# B&R Automation Studio project soft_bellows_plc
Automation Studio 4.9

## Configuration Config1

CPU 4PPC70.0702-20B, AutomationRuntime B4.93, Build 4.1.2, Safety 0.0, Vc V4.72.6

### Task classes (Cpu.sw)
```
Cyclic#1 (cycle 2000 us):
  Server <- Source.UDP.Server.prg
  Client <- Source.UDP.Client.prg
Cyclic#4 (cycle 4000 us, tolerance 80000 us):
  Program1 <- Source.Program.prg
DataObjects: Acp10sys
VcDataObjects: Visu <- Visu.dob
Binaries: FWRules, TCData, udbdef, vccdt, vccbmp, Visu03, vccline, vcfile, arial, vcrt, vccstr, vcbclass, vccbtn, vcmgr, vcgclass, vcdsint, vcptelo, vcchtml, vcpdihd, vcshared, arialbd, vcxml, vccnum, vcpdi855, vccalarm, vccurl, vccslider, vccbar, vcpfppc7, vcctext, Visu01, vcpdsw, vcfntttf, vccovl, vcalarm, Visu02, vcctrend, vcpdi815, vcdsloc, vcchspot, vctcal, vcpk, iomap, arconfig, asfw, ashwac, sysconf, User, Role, ashwd, acp10cfg, Acp10map
Libraries: Acp10man, Acp10par, NcGlobal, Acp10_MC, sys_lib, pomoc_lib, brsystem, runtime, MTLinAlg, AsTCP, AsArLog, traj_lib, regulatory, AsUDP, asstring, standard, astime, fileio, powerlnk, asieccon, vcresman, dataobj
```

### Hardware
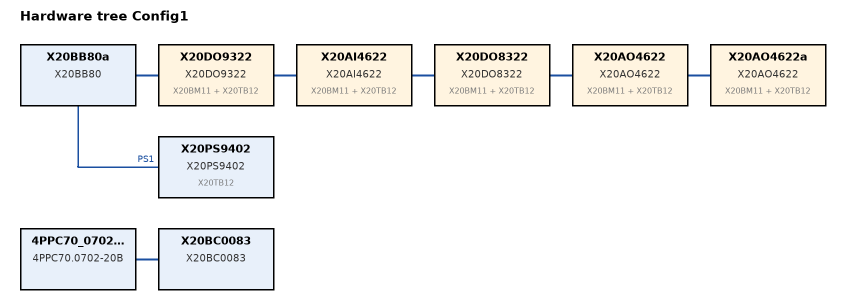
```
4PPC70_0702_20B : 4PPC70.0702-20B v1.5.4.0
  Connector IF2:
    ActivateDevice = 1
    Mode = Manual
    InternetAddress = 192.168.1.100
    SubnetMask = 255.255.255.0
    ActivateSnmp = 2
  ConfigurationID = pneuStand_Config1
  UserPartitionSize = 0
  TimerDeviceType = EPLX2X
  TimerDevice = 4PPC70_0702_20B.IF1
  TaskClassIdleTime = 2000
  Cyclic1Duration = 2000
  Cyclic3Duration = 2000
  Cyclic3Tolerance = 40000
  Cyclic4Duration = 4000
  Cyclic4Tolerance = 80000
  Cyclic5Duration = 20000
  Cyclic5Tolerance = 20000
  Cyclic6Duration = 1000000
  Cyclic6Tolerance = 1000000
  FileDevice1
  FileDeviceName1 = USER
  FileDevicePath1 = USER_PATH
  VcObjectName = Visu
  KeyMatrixPriority = HigherCyclic3
  KeyMappingFile = VC\4PPC70_0702_20B.dis
X20AI4622 : X20AI4622 v1.2.0.0  [SS1 -> X20TB12c.SS; SL -> X20BM11b.SL1]
  Supervision = off
X20AO4622 : X20AO4622 v1.3.0.0  [SS1 -> X20TB12.SS; SL -> X20BM11.SL1]
X20AO4622a : X20AO4622 v1.3.0.0  [SS1 -> X20TB12e.SS; SL -> X20BM11d.SL1]
X20BB80a : X20BB80 v1.1.0.0
X20BC0083 : X20BC0083 v2.14.0.0  [PLK1 -> 4PPC70_0702_20B.IF1 (NodeNumber=1) [Cable Type=PowerlinkCable, Length=10, Version=1.0.0.3]; SL -> X20BB80a.SL1]
  Supervision = off
X20BM11 : X20BM11 v1.1.0.0  [X2X1 -> X20BM11c.X2X2]
X20BM11a : X20BM11 v1.1.0.0  [X2X1 -> X20BB80a.IF1]
X20BM11b : X20BM11 v1.1.0.0  [X2X1 -> X20BM11a.X2X2]
X20BM11c : X20BM11 v1.1.0.0  [X2X1 -> X20BM11b.X2X2]
X20BM11d : X20BM11 v1.1.0.0  [X2X1 -> X20BM11.X2X2]
X20DO8322 : X20DO8322 v1.5.0.0  [SS1 -> X20TB12d.SS; SL -> X20BM11c.SL1]
  Supervision = off
X20DO9322 : X20DO9322 v1.5.0.0  [SS1 -> X20TB12a.SS; SL -> X20BM11a.SL1]
  Supervision = off
X20PS9402 : X20PS9402 v1.2.0.0  [SS1 -> X20TB12b.SS; PS -> X20BB80a.PS1]
  Supervision = off
X20TB12 : X20TB12 v1.0.0.0
X20TB12a : X20TB12 v1.0.0.0
X20TB12b : X20TB12 v1.0.0.0
X20TB12c : X20TB12 v1.0.0.0
X20TB12d : X20TB12 v1.0.0.0
X20TB12e : X20TB12 v1.0.0.0
```

### IoMap.iom - 4PPC70_0702_20B/IoMap.iom
```iecst
VAR_CONFIG
	::tlacidla.ventil[0] AT %QX."X20DO8322".DigitalOutput01;
	::tlacidla.ventil[1] AT %QX."X20DO8322".DigitalOutput02;
	::tlacidla.ventil[2] AT %QX."X20DO8322".DigitalOutput04;
	::tlacidla.ventil[3] AT %QX."X20DO8322".DigitalOutput05;
	::regulatory.reg[1] AT %QW."X20AO4622".AnalogOutput01;
	::regulatory.reg[2] AT %QW."X20AO4622".AnalogOutput02;
	::regulatory.reg[7] AT %QW."X20AO4622".AnalogOutput03;
	::regulatory.reg[6] AT %QW."X20AO4622".AnalogOutput04;
	::regulatory.reg[5] AT %QW."X20AO4622a".AnalogOutput01;
	::regulatory.reg[0] AT %QW."X20AO4622a".AnalogOutput02;
	::regulatory.reg[4] AT %QW."X20AO4622a".AnalogOutput03;
	::regulatory.reg[3] AT %QW."X20AO4622a".AnalogOutput04;
END_VAR
```

## Logical view

Binary libraries used (declarations not repeated): operator, runtime, astime, AsIecCon, Acp10man, Acp10par, NcGlobal, Acp10_MC, sys_lib, brsystem, MTLinAlg 5.12.0, AsArLog, AsTCP, AsUDP, asstring, standard

### Global.typ - Global data types
```iecst
TYPE
	packetUDP : 	STRUCT
		comma : INT; (*Positions of comma in received packet*)
		pStart : INT; (*Start of pressure values*)
		packet_pressure : STRING[80]; (*Full received packet*)
		length : INT; (*Length of full packet*)
		pEnd : INT; (*End of pressure values*)
		pressureString : ARRAY[0..7]OF STRING[8];
		pressureAO : ARRAY[0..7]OF REAL;
	END_STRUCT;
	Analog_input : 	STRUCT
		AI_2 : INT;
		AI_3 : INT;
		AI_4 : INT;
		AI_1 : INT;
	END_STRUCT;
	Digital_output : 	STRUCT
		DO_2 : BOOL;
		DO_3 : BOOL;
		DO_4 : BOOL;
		DO_5 : BOOL;
		DO_6 : BOOL;
		DO_7 : BOOL;
		DO_8 : BOOL;
		DO_9 : BOOL;
		DO_10 : BOOL;
		DO_11 : BOOL;
		DO_12 : BOOL;
		DO_1 : BOOL;
	END_STRUCT;
	regulators : 	STRUCT
		reg_2 : INT;
		reg_3 : INT;
		reg_4 : INT;
		reg_5 : INT;
		reg_6 : INT;
		reg_7 : INT;
		reg_8 : INT;
		reg_1 : INT;
		reg : ARRAY[0..7]OF INT;
	END_STRUCT;
	buttons : 	STRUCT
		zapni : BOOL;
		ventil : ARRAY[0..3]OF BOOL;
	END_STRUCT;
	display_variables : 	STRUCT
		in_reg : ARRAY[0..7]OF INT;
	END_STRUCT;
END_TYPE
```

### Global.var - Global variables
```iecst
VAR
	digital_output : Digital_output;
	tlacidla : buttons;
	regulatory : regulators;
	display : display_variables;
	packet : packetUDP;
	analog_input : Analog_input;
END_VAR
```

### Package Logical/Libraries - Global libraries

### Library Logical/Libraries/traj_lib (ANSIC)

#### traj_lib.typ
```iecst
TYPE
	B_generator_trajektorie_test_T :  STRUCT
		Input1 :  REAL;
		Input2 :  REAL;
		Input3 :  REAL;
		Input4 :  REAL;
		Input :  REAL;
		Gain :  ARRAY[0..299] OF REAL;
		Gain1 :  INT;
	END_STRUCT;

	tag_RTM_generator_trajektorie_T :  STRUCT
		errorStatus :  REFERENCE TO USINT;
		blockIO :  REFERENCE TO B_generator_trajektorie_test_T;
	END_STRUCT;

	RT_MODEL_generator_trajektori_T :tag_RTM_generator_trajektorie_T;	(*  *)

END_TYPE
```

#### generator_trajektorie_test.h
```c
/*
 * generator_trajektorie_test.h
 *
 * Academic License - for use in teaching, academic research, and meeting
 * course requirements at degree granting institutions only.  Not for
 * government, commercial, or other organizational use.
 *
 * Code generation for model "generator_trajektorie_test".
 *
 * Model version              : 1.23
 * Simulink Coder version : 9.6 (R2021b) 14-May-2021
 * C source code generated on : Fri Mar 25 13:28:48 2022
 *
 * Target selection: bur_grt.tlc
 * Note: GRT includes extra infrastructure and instrumentation for prototyping
 * Embedded hardware selection: Intel->x86/Pentium
 * Code generation objectives: Unspecified
 * Validation result: Not run
 */

#ifndef RTW_HEADER_generator_trajektorie_test_h_
#define RTW_HEADER_generator_trajektorie_test_h_
#include <math.h>
#include <stddef.h>
#include <string.h>
#ifndef generator_trajektorie_test_COMMON_INCLUDES_
#define generator_trajektorie_test_COMMON_INCLUDES_
#include <stdlib.h>
#include "rtwtypes.h"
#include "rtw_continuous.h"
#include "rtw_solver.h"
#endif                         /* generator_trajektorie_test_COMMON_INCLUDES_ */

#include "generator_trajektorie_test_types.h"
#include "traj_lib.h"
/* Beginning of Dynamic TypeDefs: */
/* End of Dynamic TypeDefs: */
#ifndef MIN
#define MIN(a,b)	((a) < (b) ? (a) : (b))
#endif

#ifndef MAX
#define MAX(a,b)	((a) > (b) ? (a) : (b))
#endif

#ifndef AST_ROUND
#define AST_ROUND(x) ((x)>=0?(long long)((x)+0.5):(long long)((x)-0.5))
#endif

/* Shared type includes */
#include "multiword_types.h"
#include "rtGetNaN.h"
#include "rt_nonfinite.h"
#include "rtGetInf.h"
#include "rt_defines.h"

/* Macros for accessing real-time model data structure */
#ifndef rtmGetBlockIO
#define rtmGetBlockIO(rtm)             ((rtm)->blockIO)
#endif

#ifndef rtmSetBlockIO
#define rtmSetBlockIO(rtm, val)        ((rtm)->blockIO = (val))
#endif

#ifndef rtmGetErrorStatus
#define rtmGetErrorStatus(rtm)         ((rtm)->errorStatus)
#endif

#ifndef rtmSetErrorStatus
#define rtmSetErrorStatus(rtm, val)    ((rtm)->errorStatus = (val))
#endif

#define generator_trajektorie_test_M_TYPE RT_MODEL_generator_trajektori_T

/* Block signals (default storage) */

/* Real-time Model Data Structure */

/* External data declarations for dependent source files */
extern const char *RT_MEMORY_ALLOCATION_ERROR;

/* Model entry point functions */
extern void generator_trajektorie_test_initializeMemory(RT_MODEL_generator_trajektori_T * const generator_trajektorie_test_M, struct traj* inst);
extern void generator_trajektorie_test_initialize
  (RT_MODEL_generator_trajektori_T *const generator_trajektorie_test_M, struct traj* inst);
extern void generator_trajektorie_test_step(RT_MODEL_generator_trajektori_T *
  const generator_trajektorie_test_M, struct traj* inst);
extern void generator_trajektorie_test_terminate(RT_MODEL_generator_trajektori_T
  * generator_trajektorie_test_M, struct traj* inst);

/*-
 * The generated code includes comments that allow you to trace directly
 * back to the appropriate location in the model.  The basic format
 * is <system>/block_name, where system is the system number (uniquely
 * assigned by Simulink) and block_name is the name of the block.
 *
 * Use the MATLAB hilite_system command to trace the generated code back
 * to the model.  For example,
 *
 * hilite_system('<S3>')    - opens system 3
 * hilite_system('<S3>/Kp') - opens and selects block Kp which resides in S3
 *
 * Here is the system hierarchy for this model
 *
 * '<Root>' : 'generator_trajektorie_test'
 * '<S1>'   : 'generator_trajektorie_test/MATLAB Function'
 */
#endif                            /* RTW_HEADER_generator_trajektorie_test_h_ */
```

#### generator_trajektorie_test_private.h
```c
/*
 * generator_trajektorie_test_private.h
 *
 * Academic License - for use in teaching, academic research, and meeting
 * course requirements at degree granting institutions only.  Not for
 * government, commercial, or other organizational use.
 *
 * Code generation for model "generator_trajektorie_test".
 *
 * Model version              : 1.23
 * Simulink Coder version : 9.6 (R2021b) 14-May-2021
 * C source code generated on : Fri Mar 25 13:28:48 2022
 *
 * Target selection: bur_grt.tlc
 * Note: GRT includes extra infrastructure and instrumentation for prototyping
 * Embedded hardware selection: Intel->x86/Pentium
 * Code generation objectives: Unspecified
 * Validation result: Not run
 */

#ifndef RTW_HEADER_generator_trajektorie_test_private_h_
#define RTW_HEADER_generator_trajektorie_test_private_h_
#include "rtwtypes.h"
#include "multiword_types.h"
#if !defined(rt_VALIDATE_MEMORY)
#define rt_VALIDATE_MEMORY(S, ptr)     if(!(ptr)) {\
 rtmSetErrorStatus(generator_trajektorie_test_M, RT_MEMORY_ALLOCATION_ERROR);\
 }
#endif

#if !defined(rt_FREE)
#if !defined(_WIN32)
#define rt_FREE(ptr)                   if((ptr) != (NULL)) {\
 free((ptr));\
 (ptr) = (NULL);\
 }
#else

/* Visual and other windows compilers declare free without const */
#define rt_FREE(ptr)                   if((ptr) != (NULL)) {\
 free((void *)(ptr));\
 (ptr) = (NULL);\
 }
#endif
#endif
#endif                    /* RTW_HEADER_generator_trajektorie_test_private_h_ */
```

#### generator_trajektorie_test_types.h
```c
/*
 * generator_trajektorie_test_types.h
 *
 * Academic License - for use in teaching, academic research, and meeting
 * course requirements at degree granting institutions only.  Not for
 * government, commercial, or other organizational use.
 *
 * Code generation for model "generator_trajektorie_test".
 *
 * Model version              : 1.23
 * Simulink Coder version : 9.6 (R2021b) 14-May-2021
 * C source code generated on : Fri Mar 25 13:28:48 2022
 *
 * Target selection: bur_grt.tlc
 * Note: GRT includes extra infrastructure and instrumentation for prototyping
 * Embedded hardware selection: Intel->x86/Pentium
 * Code generation objectives: Unspecified
 * Validation result: Not run
 */

#ifndef RTW_HEADER_generator_trajektorie_test_types_h_
#define RTW_HEADER_generator_trajektorie_test_types_h_

/* Model Code Variants */

/* Forward declaration for rtModel */

#endif                      /* RTW_HEADER_generator_trajektorie_test_types_h_ */
```

#### multiword_types.h
```c
/*
 * multiword_types.h
 *
 * Academic License - for use in teaching, academic research, and meeting
 * course requirements at degree granting institutions only.  Not for
 * government, commercial, or other organizational use.
 *
 * Code generation for model "generator_trajektorie_test".
 *
 * Model version              : 1.23
 * Simulink Coder version : 9.6 (R2021b) 14-May-2021
 * C source code generated on : Fri Mar 25 13:28:48 2022
 *
 * Target selection: bur_grt.tlc
 * Note: GRT includes extra infrastructure and instrumentation for prototyping
 * Embedded hardware selection: Intel->x86/Pentium
 * Code generation objectives: Unspecified
 * Validation result: Not run
 */

#ifndef MULTIWORD_TYPES_H
#define MULTIWORD_TYPES_H
#include "rtwtypes.h"

/*
 * MultiWord supporting definitions
 */
typedef long int long_T;

/*
 * MultiWord types
 */
typedef struct {
  uint32_T chunks[2];
} int64m_T;

typedef struct {
  int64m_T re;
  int64m_T im;
} cint64m_T;

typedef struct {
  uint32_T chunks[2];
} uint64m_T;

typedef struct {
  uint64m_T re;
  uint64m_T im;
} cuint64m_T;

typedef struct {
  uint32_T chunks[3];
} int96m_T;

typedef struct {
  int96m_T re;
  int96m_T im;
} cint96m_T;

typedef struct {
  uint32_T chunks[3];
} uint96m_T;

typedef struct {
  uint96m_T re;
  uint96m_T im;
} cuint96m_T;

typedef struct {
  uint32_T chunks[4];
} int128m_T;

typedef struct {
  int128m_T re;
  int128m_T im;
} cint128m_T;

typedef struct {
  uint32_T chunks[4];
} uint128m_T;

typedef struct {
  uint128m_T re;
  uint128m_T im;
} cuint128m_T;

typedef struct {
  uint32_T chunks[5];
} int160m_T;

typedef struct {
  int160m_T re;
  int160m_T im;
} cint160m_T;

typedef struct {
  uint32_T chunks[5];
} uint160m_T;

typedef struct {
  uint160m_T re;
  uint160m_T im;
} cuint160m_T;

typedef struct {
  uint32_T chunks[6];
} int192m_T;

typedef struct {
  int192m_T re;
  int192m_T im;
} cint192m_T;

typedef struct {
  uint32_T chunks[6];
} uint192m_T;

typedef struct {
  uint192m_T re;
  uint192m_T im;
} cuint192m_T;

typedef struct {
  uint32_T chunks[7];
} int224m_T;

typedef struct {
  int224m_T re;
  int224m_T im;
} cint224m_T;

typedef struct {
  uint32_T chunks[7];
} uint224m_T;

typedef struct {
  uint224m_T re;
  uint224m_T im;
} cuint224m_T;

typedef struct {
  uint32_T chunks[8];
} int256m_T;

typedef struct {
  int256m_T re;
  int256m_T im;
} cint256m_T;

typedef struct {
  uint32_T chunks[8];
} uint256m_T;

typedef struct {
  uint256m_T re;
  uint256m_T im;
} cuint256m_T;

typedef struct {
  uint32_T chunks[9];
} int288m_T;

typedef struct {
  int288m_T re;
  int288m_T im;
} cint288m_T;

typedef struct {
  uint32_T chunks[9];
} uint288m_T;

typedef struct {
  uint288m_T re;
  uint288m_T im;
} cuint288m_T;

typedef struct {
  uint32_T chunks[10];
} int320m_T;

typedef struct {
  int320m_T re;
  int320m_T im;
} cint320m_T;

typedef struct {
  uint32_T chunks[10];
} uint320m_T;

typedef struct {
  uint320m_T re;
  uint320m_T im;
} cuint320m_T;

typedef struct {
  uint32_T chunks[11];
} int352m_T;

typedef struct {
  int352m_T re;
  int352m_T im;
} cint352m_T;

typedef struct {
  uint32_T chunks[11];
} uint352m_T;

typedef struct {
  uint352m_T re;
  uint352m_T im;
} cuint352m_T;

typedef struct {
  uint32_T chunks[12];
} int384m_T;

typedef struct {
  int384m_T re;
  int384m_T im;
} cint384m_T;

typedef struct {
  uint32_T chunks[12];
} uint384m_T;

typedef struct {
  uint384m_T re;
  uint384m_T im;
} cuint384m_T;

typedef struct {
  uint32_T chunks[13];
} int416m_T;

typedef struct {
  int416m_T re;
  int416m_T im;
} cint416m_T;

typedef struct {
  uint32_T chunks[13];
} uint416m_T;

typedef struct {
  uint416m_T re;
  uint416m_T im;
} cuint416m_T;

typedef struct {
  uint32_T chunks[14];
} int448m_T;

typedef struct {
  int448m_T re;
  int448m_T im;
} cint448m_T;

typedef struct {
  uint32_T chunks[14];
} uint448m_T;

typedef struct {
  uint448m_T re;
  uint448m_T im;
} cuint448m_T;

typedef struct {
  uint32_T chunks[15];
} int480m_T;

typedef struct {
  int480m_T re;
  int480m_T im;
} cint480m_T;

typedef struct {
  uint32_T chunks[15];
} uint480m_T;

typedef struct {
  uint480m_T re;
  uint480m_T im;
} cuint480m_T;

typedef struct {
  uint32_T chunks[16];
} int512m_T;

typedef struct {
  int512m_T re;
  int512m_T im;
} cint512m_T;

typedef struct {
  uint32_T chunks[16];
} uint512m_T;

typedef struct {
  uint512m_T re;
  uint512m_T im;
} cuint512m_T;

typedef struct {
  uint32_T chunks[17];
} int544m_T;

typedef struct {
  int544m_T re;
  int544m_T im;
} cint544m_T;

typedef struct {
  uint32_T chunks[17];
} uint544m_T;

typedef struct {
  uint544m_T re;
  uint544m_T im;
} cuint544m_T;

typedef struct {
  uint32_T chunks[18];
} int576m_T;

typedef struct {
  int576m_T re;
  int576m_T im;
} cint576m_T;

typedef struct {
  uint32_T chunks[18];
} uint576m_T;

typedef struct {
  uint576m_T re;
  uint576m_T im;
} cuint576m_T;

typedef struct {
  uint32_T chunks[19];
} int608m_T;

typedef struct {
  int608m_T re;
  int608m_T im;
} cint608m_T;

typedef struct {
  uint32_T chunks[19];
} uint608m_T;

typedef struct {
  uint608m_T re;
  uint608m_T im;
} cuint608m_T;

typedef struct {
  uint32_T chunks[20];
} int640m_T;

typedef struct {
  int640m_T re;
  int640m_T im;
} cint640m_T;

typedef struct {
  uint32_T chunks[20];
} uint640m_T;

typedef struct {
  uint640m_T re;
  uint640m_T im;
} cuint640m_T;

typedef struct {
  uint32_T chunks[21];
} int672m_T;

typedef struct {
  int672m_T re;
  int672m_T im;
} cint672m_T;

typedef struct {
  uint32_T chunks[21];
} uint672m_T;

typedef struct {
  uint672m_T re;
  uint672m_T im;
} cuint672m_T;

typedef struct {
  uint32_T chunks[22];
} int704m_T;

typedef struct {
  int704m_T re;
  int704m_T im;
} cint704m_T;

typedef struct {
  uint32_T chunks[22];
} uint704m_T;

typedef struct {
  uint704m_T re;
  uint704m_T im;
} cuint704m_T;

typedef struct {
  uint32_T chunks[23];
} int736m_T;

typedef struct {
  int736m_T re;
  int736m_T im;
} cint736m_T;

typedef struct {
  uint32_T chunks[23];
} uint736m_T;

typedef struct {
  uint736m_T re;
  uint736m_T im;
} cuint736m_T;

typedef struct {
  uint32_T chunks[24];
} int768m_T;

typedef struct {
  int768m_T re;
  int768m_T im;
} cint768m_T;

typedef struct {
  uint32_T chunks[24];
} uint768m_T;

typedef struct {
  uint768m_T re;
  uint768m_T im;
} cuint768m_T;

typedef struct {
  uint32_T chunks[25];
} int800m_T;

typedef struct {
  int800m_T re;
  int800m_T im;
} cint800m_T;

typedef struct {
  uint32_T chunks[25];
} uint800m_T;

typedef struct {
  uint800m_T re;
  uint800m_T im;
} cuint800m_T;

typedef struct {
  uint32_T chunks[26];
} int832m_T;

typedef struct {
  int832m_T re;
  int832m_T im;
} cint832m_T;

typedef struct {
  uint32_T chunks[26];
} uint832m_T;

typedef struct {
  uint832m_T re;
  uint832m_T im;
} cuint832m_T;

typedef struct {
  uint32_T chunks[27];
} int864m_T;

typedef struct {
  int864m_T re;
  int864m_T im;
} cint864m_T;

typedef struct {
  uint32_T chunks[27];
} uint864m_T;

typedef struct {
  uint864m_T re;
  uint864m_T im;
} cuint864m_T;

typedef struct {
  uint32_T chunks[28];
} int896m_T;

typedef struct {
  int896m_T re;
  int896m_T im;
} cint896m_T;

typedef struct {
  uint32_T chunks[28];
} uint896m_T;

typedef struct {
  uint896m_T re;
  uint896m_T im;
} cuint896m_T;

typedef struct {
  uint32_T chunks[29];
} int928m_T;

typedef struct {
  int928m_T re;
  int928m_T im;
} cint928m_T;

typedef struct {
  uint32_T chunks[29];
} uint928m_T;

typedef struct {
  uint928m_T re;
  uint928m_T im;
} cuint928m_T;

typedef struct {
  uint32_T chunks[30];
} int960m_T;

typedef struct {
  int960m_T re;
  int960m_T im;
} cint960m_T;

typedef struct {
  uint32_T chunks[30];
} uint960m_T;

typedef struct {
  uint960m_T re;
  uint960m_T im;
} cuint960m_T;

typedef struct {
  uint32_T chunks[31];
} int992m_T;

typedef struct {
  int992m_T re;
  int992m_T im;
} cint992m_T;

typedef struct {
  uint32_T chunks[31];
} uint992m_T;

typedef struct {
  uint992m_T re;
  uint992m_T im;
} cuint992m_T;

typedef struct {
  uint32_T chunks[32];
} int1024m_T;

typedef struct {
  int1024m_T re;
  int1024m_T im;
} cint1024m_T;

typedef struct {
  uint32_T chunks[32];
} uint1024m_T;

typedef struct {
  uint1024m_T re;
  uint1024m_T im;
} cuint1024m_T;

typedef struct {
  uint32_T chunks[33];
} int1056m_T;

typedef struct {
  int1056m_T re;
  int1056m_T im;
} cint1056m_T;

typedef struct {
  uint32_T chunks[33];
} uint1056m_T;

typedef struct {
  uint1056m_T re;
  uint1056m_T im;
} cuint1056m_T;

typedef struct {
  uint32_T chunks[34];
} int1088m_T;

typedef struct {
  int1088m_T re;
  int1088m_T im;
} cint1088m_T;

typedef struct {
  uint32_T chunks[34];
} uint1088m_T;

typedef struct {
  uint1088m_T re;
  uint1088m_T im;
} cuint1088m_T;

typedef struct {
  uint32_T chunks[35];
} int1120m_T;

typedef struct {
  int1120m_T re;
  int1120m_T im;
} cint1120m_T;

typedef struct {
  uint32_T chunks[35];
} uint1120m_T;

typedef struct {
  uint1120m_T re;
  uint1120m_T im;
} cuint1120m_T;

typedef struct {
  uint32_T chunks[36];
} int1152m_T;

typedef struct {
  int1152m_T re;
  int1152m_T im;
} cint1152m_T;

typedef struct {
  uint32_T chunks[36];
} uint1152m_T;

typedef struct {
  uint1152m_T re;
  uint1152m_T im;
} cuint1152m_T;

typedef struct {
  uint32_T chunks[37];
} int1184m_T;

typedef struct {
  int1184m_T re;
  int1184m_T im;
} cint1184m_T;

typedef struct {
  uint32_T chunks[37];
} uint1184m_T;

typedef struct {
  uint1184m_T re;
  uint1184m_T im;
} cuint1184m_T;

typedef struct {
  uint32_T chunks[38];
} int1216m_T;

typedef struct {
  int1216m_T re;
  int1216m_T im;
} cint1216m_T;

typedef struct {
  uint32_T chunks[38];
} uint1216m_T;

typedef struct {
  uint1216m_T re;
  uint1216m_T im;
} cuint1216m_T;

typedef struct {
  uint32_T chunks[39];
} int1248m_T;

typedef struct {
  int1248m_T re;
  int1248m_T im;
} cint1248m_T;

typedef struct {
  uint32_T chunks[39];
} uint1248m_T;

typedef struct {
  uint1248m_T re;
  uint1248m_T im;
} cuint1248m_T;

typedef struct {
  uint32_T chunks[40];
} int1280m_T;

typedef struct {
  int1280m_T re;
  int1280m_T im;
} cint1280m_T;

typedef struct {
  uint32_T chunks[40];
} uint1280m_T;

typedef struct {
  uint1280m_T re;
  uint1280m_T im;
} cuint1280m_T;

typedef struct {
  uint32_T chunks[41];
} int1312m_T;

typedef struct {
  int1312m_T re;
  int1312m_T im;
} cint1312m_T;

typedef struct {
  uint32_T chunks[41];
} uint1312m_T;

typedef struct {
  uint1312m_T re;
  uint1312m_T im;
} cuint1312m_T;

typedef struct {
  uint32_T chunks[42];
} int1344m_T;

typedef struct {
  int1344m_T re;
  int1344m_T im;
} cint1344m_T;

typedef struct {
  uint32_T chunks[42];
} uint1344m_T;

typedef struct {
  uint1344m_T re;
  uint1344m_T im;
} cuint1344m_T;

typedef struct {
  uint32_T chunks[43];
} int1376m_T;

typedef struct {
  int1376m_T re;
  int1376m_T im;
} cint1376m_T;

typedef struct {
  uint32_T chunks[43];
} uint1376m_T;

typedef struct {
  uint1376m_T re;
  uint1376m_T im;
} cuint1376m_T;

typedef struct {
  uint32_T chunks[44];
} int1408m_T;

typedef struct {
  int1408m_T re;
  int1408m_T im;
} cint1408m_T;

typedef struct {
  uint32_T chunks[44];
} uint1408m_T;

typedef struct {
  uint1408m_T re;
  uint1408m_T im;
} cuint1408m_T;

typedef struct {
  uint32_T chunks[45];
} int1440m_T;

typedef struct {
  int1440m_T re;
  int1440m_T im;
} cint1440m_T;

typedef struct {
  uint32_T chunks[45];
} uint1440m_T;

typedef struct {
  uint1440m_T re;
  uint1440m_T im;
} cuint1440m_T;

typedef struct {
  uint32_T chunks[46];
} int1472m_T;

typedef struct {
  int1472m_T re;
  int1472m_T im;
} cint1472m_T;

typedef struct {
  uint32_T chunks[46];
} uint1472m_T;

typedef struct {
  uint1472m_T re;
  uint1472m_T im;
} cuint1472m_T;

typedef struct {
  uint32_T chunks[47];
} int1504m_T;

typedef struct {
  int1504m_T re;
  int1504m_T im;
} cint1504m_T;

typedef struct {
  uint32_T chunks[47];
} uint1504m_T;

typedef struct {
  uint1504m_T re;
  uint1504m_T im;
} cuint1504m_T;

typedef struct {
  uint32_T chunks[48];
} int1536m_T;

typedef struct {
  int1536m_T re;
  int1536m_T im;
} cint1536m_T;

typedef struct {
  uint32_T chunks[48];
} uint1536m_T;

typedef struct {
  uint1536m_T re;
  uint1536m_T im;
} cuint1536m_T;

typedef struct {
  uint32_T chunks[49];
} int1568m_T;

typedef struct {
  int1568m_T re;
  int1568m_T im;
} cint1568m_T;

typedef struct {
  uint32_T chunks[49];
} uint1568m_T;

typedef struct {
  uint1568m_T re;
  uint1568m_T im;
} cuint1568m_T;

typedef struct {
  uint32_T chunks[50];
} int1600m_T;

typedef struct {
  int1600m_T re;
  int1600m_T im;
} cint1600m_T;

typedef struct {
  uint32_T chunks[50];
} uint1600m_T;

typedef struct {
  uint1600m_T re;
  uint1600m_T im;
} cuint1600m_T;

typedef struct {
  uint32_T chunks[51];
} int1632m_T;

typedef struct {
  int1632m_T re;
  int1632m_T im;
} cint1632m_T;

typedef struct {
  uint32_T chunks[51];
} uint1632m_T;

typedef struct {
  uint1632m_T re;
  uint1632m_T im;
} cuint1632m_T;

typedef struct {
  uint32_T chunks[52];
} int1664m_T;

typedef struct {
  int1664m_T re;
  int1664m_T im;
} cint1664m_T;

typedef struct {
  uint32_T chunks[52];
} uint1664m_T;

typedef struct {
  uint1664m_T re;
  uint1664m_T im;
} cuint1664m_T;

typedef struct {
  uint32_T chunks[53];
} int1696m_T;

typedef struct {
  int1696m_T re;
  int1696m_T im;
} cint1696m_T;

typedef struct {
  uint32_T chunks[53];
} uint1696m_T;

typedef struct {
  uint1696m_T re;
  uint1696m_T im;
} cuint1696m_T;

typedef struct {
  uint32_T chunks[54];
} int1728m_T;

typedef struct {
  int1728m_T re;
  int1728m_T im;
} cint1728m_T;

typedef struct {
  uint32_T chunks[54];
} uint1728m_T;

typedef struct {
  uint1728m_T re;
  uint1728m_T im;
} cuint1728m_T;

typedef struct {
  uint32_T chunks[55];
} int1760m_T;

typedef struct {
  int1760m_T re;
  int1760m_T im;
} cint1760m_T;

typedef struct {
  uint32_T chunks[55];
} uint1760m_T;

typedef struct {
  uint1760m_T re;
  uint1760m_T im;
} cuint1760m_T;

typedef struct {
  uint32_T chunks[56];
} int1792m_T;

typedef struct {
  int1792m_T re;
  int1792m_T im;
} cint1792m_T;

typedef struct {
  uint32_T chunks[56];
} uint1792m_T;

typedef struct {
  uint1792m_T re;
  uint1792m_T im;
} cuint1792m_T;

typedef struct {
  uint32_T chunks[57];
} int1824m_T;

typedef struct {
  int1824m_T re;
  int1824m_T im;
} cint1824m_T;

typedef struct {
  uint32_T chunks[57];
} uint1824m_T;

typedef struct {
  uint1824m_T re;
  uint1824m_T im;
} cuint1824m_T;

typedef struct {
  uint32_T chunks[58];
} int1856m_T;

typedef struct {
  int1856m_T re;
  int1856m_T im;
} cint1856m_T;

typedef struct {
  uint32_T chunks[58];
} uint1856m_T;

typedef struct {
  uint1856m_T re;
  uint1856m_T im;
} cuint1856m_T;

typedef struct {
  uint32_T chunks[59];
} int1888m_T;

typedef struct {
  int1888m_T re;
  int1888m_T im;
} cint1888m_T;

typedef struct {
  uint32_T chunks[59];
} uint1888m_T;

typedef struct {
  uint1888m_T re;
  uint1888m_T im;
} cuint1888m_T;

typedef struct {
  uint32_T chunks[60];
} int1920m_T;

typedef struct {
  int1920m_T re;
  int1920m_T im;
} cint1920m_T;

typedef struct {
  uint32_T chunks[60];
} uint1920m_T;

typedef struct {
  uint1920m_T re;
  uint1920m_T im;
} cuint1920m_T;

typedef struct {
  uint32_T chunks[61];
} int1952m_T;

typedef struct {
  int1952m_T re;
  int1952m_T im;
} cint1952m_T;

typedef struct {
  uint32_T chunks[61];
} uint1952m_T;

typedef struct {
  uint1952m_T re;
  uint1952m_T im;
} cuint1952m_T;

typedef struct {
  uint32_T chunks[62];
} int1984m_T;

typedef struct {
  int1984m_T re;
  int1984m_T im;
} cint1984m_T;

typedef struct {
  uint32_T chunks[62];
} uint1984m_T;

typedef struct {
  uint1984m_T re;
  uint1984m_T im;
} cuint1984m_T;

typedef struct {
  uint32_T chunks[63];
} int2016m_T;

typedef struct {
  int2016m_T re;
  int2016m_T im;
} cint2016m_T;

typedef struct {
  uint32_T chunks[63];
} uint2016m_T;

typedef struct {
  uint2016m_T re;
  uint2016m_T im;
} cuint2016m_T;

typedef struct {
  uint32_T chunks[64];
} int2048m_T;

typedef struct {
  int2048m_T re;
  int2048m_T im;
} cint2048m_T;

typedef struct {
  uint32_T chunks[64];
} uint2048m_T;

typedef struct {
  uint2048m_T re;
  uint2048m_T im;
} cuint2048m_T;

#endif                                 /* MULTIWORD_TYPES_H */
```

#### rt_defines.h
```c
/*
 * rt_defines.h
 *
 * Academic License - for use in teaching, academic research, and meeting
 * course requirements at degree granting institutions only.  Not for
 * government, commercial, or other organizational use.
 *
 * Code generation for model "generator_trajektorie_test".
 *
 * Model version              : 1.23
 * Simulink Coder version : 9.6 (R2021b) 14-May-2021
 * C source code generated on : Fri Mar 25 13:28:48 2022
 *
 * Target selection: bur_grt.tlc
 * Note: GRT includes extra infrastructure and instrumentation for prototyping
 * Embedded hardware selection: Intel->x86/Pentium
 * Code generation objectives: Unspecified
 * Validation result: Not run
 */

#ifndef RTW_HEADER_rt_defines_h_
#define RTW_HEADER_rt_defines_h_

/*===========*
 * Constants *
 *===========*/
#define RT_PI                          3.14159265358979323846
#define RT_PIF                         3.1415927F
#define RT_LN_10                       2.30258509299404568402
#define RT_LN_10F                      2.3025851F
#define RT_LOG10E                      0.43429448190325182765
#define RT_LOG10EF                     0.43429449F
#define RT_E                           2.7182818284590452354
#define RT_EF                          2.7182817F

/*
 * UNUSED_PARAMETER(x)
 *   Used to specify that a function parameter (argument) is required but not
 *   accessed by the function body.
 */
#ifndef UNUSED_PARAMETER
#if defined(__LCC__)
#define UNUSED_PARAMETER(x)                                      /* do nothing */
#else

/*
 * This is the semi-ANSI standard way of indicating that an
 * unused function parameter is required.
 */
#define UNUSED_PARAMETER(x)            (void) (x)
#endif
#endif
#endif                                 /* RTW_HEADER_rt_defines_h_ */
```

#### rtGetInf.h
```c
/*
 * rtGetInf.h
 *
 * Academic License - for use in teaching, academic research, and meeting
 * course requirements at degree granting institutions only.  Not for
 * government, commercial, or other organizational use.
 *
 * Code generation for model "generator_trajektorie_test".
 *
 * Model version              : 1.23
 * Simulink Coder version : 9.6 (R2021b) 14-May-2021
 * C source code generated on : Fri Mar 25 13:28:48 2022
 *
 * Target selection: bur_grt.tlc
 * Note: GRT includes extra infrastructure and instrumentation for prototyping
 * Embedded hardware selection: Intel->x86/Pentium
 * Code generation objectives: Unspecified
 * Validation result: Not run
 */

#ifndef RTW_HEADER_rtGetInf_h_
#define RTW_HEADER_rtGetInf_h_
#include <stddef.h>
#include "rtwtypes.h"
#include "rt_nonfinite.h"

extern real_T rtGetInf(void);
extern real32_T rtGetInfF(void);
extern real_T rtGetMinusInf(void);
extern real32_T rtGetMinusInfF(void);

#endif                                 /* RTW_HEADER_rtGetInf_h_ */
```

#### rtmodel.h
```c
/*
 *  rtmodel.h:
 *
 * Academic License - for use in teaching, academic research, and meeting
 * course requirements at degree granting institutions only.  Not for
 * government, commercial, or other organizational use.
 *
 * Code generation for model "generator_trajektorie_test".
 *
 * Model version              : 1.3
 * Simulink Coder version : 9.6 (R2021b) 14-May-2021
 * C source code generated on : Wed Mar  2 13:13:15 2022
 *
 * Target selection: bur_grt.tlc
 * Note: GRT includes extra infrastructure and instrumentation for prototyping
 * Embedded hardware selection: Intel->x86/Pentium
 * Code generation objectives: Unspecified
 * Validation result: Not run
 */

#ifndef RTW_HEADER_rtmodel_h_
#define RTW_HEADER_rtmodel_h_

/*
 *  Includes the appropriate headers when we are using rtModel
 */
#include "generator_trajektorie_test.h"
#define GRTINTERFACE                   0

/*
 * ROOT_IO_FORMAT: 0 (Individual arguments)
 * ROOT_IO_FORMAT: 1 (Structure reference)
 * ROOT_IO_FORMAT: 2 (Part of model data structure)
 */
#define ROOT_IO_FORMAT                 2

/* Macros generated for backwards compatibility  */
#ifndef rtmGetStopRequested
#define rtmGetStopRequested(rtm)       ((void*) 0)
#endif
#endif                                 /* RTW_HEADER_rtmodel_h_ */
```

#### lib_properties.txt
```
For manual assignment to hardware configuration please
add the following additional include directories:

\Logical\MATLAB_includes\R2021b\

And the following additional build options:

-lm -D RT_MALLOC -D MODEL=generator_trajektorie_test -D NUMST=1 -D NCSTATES=0 -D HAVESTDIO -D RT -D USE_RTMODEL -D CLASSIC_INTERFACE=0 -D ALLOCATIONFCN=1 -D TID01EQ=0 -D MAT_FILE=0 -D ONESTEPFCN=1 -D TERMFCN=1 -D MULTI_INSTANCE_CODE=1 -D INTEGER_CODE=0 -D MT=0
```

#### rtGetNaN.c
```c
/*
 * rtGetNaN.c
 *
 * Academic License - for use in teaching, academic research, and meeting
 * course requirements at degree granting institutions only.  Not for
 * government, commercial, or other organizational use.
 *
 * Code generation for model "generator_trajektorie_test".
 *
 * Model version              : 1.23
 * Simulink Coder version : 9.6 (R2021b) 14-May-2021
 * C source code generated on : Fri Mar 25 13:28:48 2022
 *
 * Target selection: bur_grt.tlc
 * Note: GRT includes extra infrastructure and instrumentation for prototyping
 * Embedded hardware selection: Intel->x86/Pentium
 * Code generation objectives: Unspecified
 * Validation result: Not run
 */

/*
 * Abstract:
 *      Function to initialize non-finite, NaN
 */
#include "rtGetNaN.h"
#define NumBitsPerChar                 8U

/*
 * Initialize rtNaN needed by the generated code.
 * NaN is initialized as non-signaling. Assumes IEEE.
 */
real_T rtGetNaN(void)
{
  size_t bitsPerReal = sizeof(real_T) * (NumBitsPerChar);
  real_T nan = 0.0;
  if (bitsPerReal == 32U) {
    nan = rtGetNaNF();
  } else {
    uint16_T one = 1U;
    enum {
      LittleEndian,
      BigEndian
    } machByteOrder = (*((uint8_T *) &one) == 1U) ? LittleEndian : BigEndian;
    switch (machByteOrder) {
     case LittleEndian:
      {
        union {
          LittleEndianIEEEDouble bitVal;
          real_T fltVal;
        } tmpVal;

        tmpVal.bitVal.words.wordH = 0xFFF80000U;
        tmpVal.bitVal.words.wordL = 0x00000000U;
        nan = tmpVal.fltVal;
        break;
      }

     case BigEndian:
      {
        union {
          BigEndianIEEEDouble bitVal;
          real_T fltVal;
        } tmpVal;

        tmpVal.bitVal.words.wordH = 0x7FFFFFFFU;
        tmpVal.bitVal.words.wordL = 0xFFFFFFFFU;
        nan = tmpVal.fltVal;
        break;
      }
    }
  }

  return nan;
}

/*
 * Initialize rtNaNF needed by the generated code.
 * NaN is initialized as non-signaling. Assumes IEEE.
 */
real32_T rtGetNaNF(void)
{
  IEEESingle nanF = { { 0.0F } };

  uint16_T one = 1U;
  enum {
    LittleEndian,
    BigEndian
  } machByteOrder = (*((uint8_T *) &one) == 1U) ? LittleEndian : BigEndian;
  switch (machByteOrder) {
   case LittleEndian:
    {
      nanF.wordL.wordLuint = 0xFFC00000U;
      break;
    }

   case BigEndian:
    {
      nanF.wordL.wordLuint = 0x7FFFFFFFU;
      break;
    }
  }

  return nanF.wordL.wordLreal;
}
```

### Library Logical/Libraries/pomoc_lib (ANSIC, version 1.00.0)

#### cyklovac_BB_private.h
```c
/*
 * cyklovac_BB_private.h
 *
 * Academic License - for use in teaching, academic research, and meeting
 * course requirements at degree granting institutions only.  Not for
 * government, commercial, or other organizational use.
 *
 * Code generation for model "cyklovac_BB".
 *
 * Model version              : 1.8
 * Simulink Coder version : 9.6 (R2021b) 14-May-2021
 * C source code generated on : Thu Mar 17 07:18:42 2022
 *
 * Target selection: bur_grt.tlc
 * Note: GRT includes extra infrastructure and instrumentation for prototyping
 * Embedded hardware selection: Intel->x86/Pentium
 * Code generation objectives: Unspecified
 * Validation result: Not run
 */

#ifndef RTW_HEADER_cyklovac_BB_private_h_
#define RTW_HEADER_cyklovac_BB_private_h_
#include "rtwtypes.h"
#include "multiword_types.h"
#if !defined(rt_VALIDATE_MEMORY)
#define rt_VALIDATE_MEMORY(S, ptr)     if(!(ptr)) {\
 rtmSetErrorStatus(cyklovac_BB_M, RT_MEMORY_ALLOCATION_ERROR);\
 }
#endif

#if !defined(rt_FREE)
#if !defined(_WIN32)
#define rt_FREE(ptr)                   if((ptr) != (NULL)) {\
 free((ptr));\
 (ptr) = (NULL);\
 }
#else

/* Visual and other windows compilers declare free without const */
#define rt_FREE(ptr)                   if((ptr) != (NULL)) {\
 free((void *)(ptr));\
 (ptr) = (NULL);\
 }
#endif
#endif
#endif                                 /* RTW_HEADER_cyklovac_BB_private_h_ */
```

#### cyklovac_b.c
```c
/********************************************************************
 * COPYRIGHT -- B&R Industrial Automation GmbH
 ********************************************************************
 * Program: pomoc_lib
 * File: pomoc_lib.c
 * Author: MartinV
 * Last modified by: MartinV
 * Created: 17-Mar-2022 07:18:45
 * Last modified: Thu Mar 17 07:18:38 2022
 * Model Version: 1.8
 * Description:
 * modified Comment:
 ********************************************************************
 * Implementation of program pomoc_lib
 ********************************************************************
 * Generated with B&R Automation Studio Target for Simulink V6.5
 * (GRT based)
 ********************************************************************/

#include <bur/plctypes.h>

#include "rtwtypes.h"
#include "rtmodel.h"

#define EXPAND_CONCAT(name1,name2) name1 ## name2
#define CONCAT(name1,name2) EXPAND_CONCAT(name1,name2)
#define RT_MODEL            CONCAT(MODEL,_rtModel)

#ifdef __cplusplus

extern "C" {

#endif

/* Defines */
#define SS_TERMINATE 4
#define SS_OUTPUT 3
#define SS_INITIALIZE 2

#ifdef __cplusplus

}

#endif

#ifdef __cplusplus
    unsigned long bur_heap_size = 6553500;
#endif

void cyklovac_b(struct cyklovac_b* inst)
{
  tag_RTM_cyklovac_BB_T* const cyklovac_BB_M = &(inst)->bur_cyklovac_BB;
	inst->bur_cyklovac_BB.blockIO = &(inst)->bur_B_cyklovac_BB_T;

  switch (inst->ssMethodType)
  {
    case SS_INITIALIZE:

      /* call model initialize functions */
		/*memInit function */
		cyklovac_BB_initializeMemory(cyklovac_BB_M, inst);
		cyklovac_BB_initialize(cyklovac_BB_M, inst);
      break;

    case SS_OUTPUT:
      /* call model step functions */
		cyklovac_BB_step(cyklovac_BB_M, inst);
      break;

    case SS_TERMINATE:
      /* call model terminate function */
		cyklovac_BB_terminate(cyklovac_BB_M, inst);
	  break;
  }
}

/*****************************************************************************
   Function block sample time: 0.008
 *****************************************************************************/

/*****************************************************************************
   B&R Automation Studio Target for Simulink Version: V6.5.1 (03-Dec-2021)
 *****************************************************************************/
```

#### pomoc_lib.typ
```iecst
TYPE
B_cyklovac_BB_T : STRUCT
	Input : REAL;
	Gain : REAL;
	Gain1 : REAL;
	Gain2 : REAL;
END_STRUCT;
ConstP_cyklovac_BB_T : STRUCT
	Constant_Value : ARRAY[0..2351] OF LREAL;
END_STRUCT;
tag_RTM_cyklovac_BB_T : STRUCT
	errorStatus : REFERENCE TO USINT;
	blockIO : REFERENCE TO B_cyklovac_BB_T;
END_STRUCT;
RT_MODEL_cyklovac_BB_T : tag_RTM_cyklovac_BB_T;

END_TYPE
TYPE
END_TYPE
```

#### rt_defines.h
```c
/*
 * rt_defines.h
 *
 * Academic License - for use in teaching, academic research, and meeting
 * course requirements at degree granting institutions only.  Not for
 * government, commercial, or other organizational use.
 *
 * Code generation for model "cyklovac_BB".
 *
 * Model version              : 1.8
 * Simulink Coder version : 9.6 (R2021b) 14-May-2021
 * C source code generated on : Thu Mar 17 07:18:42 2022
 *
 * Target selection: bur_grt.tlc
 * Note: GRT includes extra infrastructure and instrumentation for prototyping
 * Embedded hardware selection: Intel->x86/Pentium
 * Code generation objectives: Unspecified
 * Validation result: Not run
 */

#ifndef RTW_HEADER_rt_defines_h_
#define RTW_HEADER_rt_defines_h_

/*===========*
 * Constants *
 *===========*/
#define RT_PI                          3.14159265358979323846
#define RT_PIF                         3.1415927F
#define RT_LN_10                       2.30258509299404568402
#define RT_LN_10F                      2.3025851F
#define RT_LOG10E                      0.43429448190325182765
#define RT_LOG10EF                     0.43429449F
#define RT_E                           2.7182818284590452354
#define RT_EF                          2.7182817F

/*
 * UNUSED_PARAMETER(x)
 *   Used to specify that a function parameter (argument) is required but not
 *   accessed by the function body.
 */
#ifndef UNUSED_PARAMETER
#if defined(__LCC__)
#define UNUSED_PARAMETER(x)                                      /* do nothing */
#else

/*
 * This is the semi-ANSI standard way of indicating that an
 * unused function parameter is required.
 */
#define UNUSED_PARAMETER(x)            (void) (x)
#endif
#endif
#endif                                 /* RTW_HEADER_rt_defines_h_ */
```

#### rtmodel.h
```c
/*
 *  rtmodel.h:
 *
 * Academic License - for use in teaching, academic research, and meeting
 * course requirements at degree granting institutions only.  Not for
 * government, commercial, or other organizational use.
 *
 * Code generation for model "cyklovac_BB".
 *
 * Model version              : 1.8
 * Simulink Coder version : 9.6 (R2021b) 14-May-2021
 * C source code generated on : Thu Mar 17 07:18:42 2022
 *
 * Target selection: bur_grt.tlc
 * Note: GRT includes extra infrastructure and instrumentation for prototyping
 * Embedded hardware selection: Intel->x86/Pentium
 * Code generation objectives: Unspecified
 * Validation result: Not run
 */

#ifndef RTW_HEADER_rtmodel_h_
#define RTW_HEADER_rtmodel_h_

/*
 *  Includes the appropriate headers when we are using rtModel
 */
#include "cyklovac_BB.h"
#define GRTINTERFACE                   0

/*
 * ROOT_IO_FORMAT: 0 (Individual arguments)
 * ROOT_IO_FORMAT: 1 (Structure reference)
 * ROOT_IO_FORMAT: 2 (Part of model data structure)
 */
#define ROOT_IO_FORMAT                 2

/* Macros generated for backwards compatibility  */
#ifndef rtmGetStopRequested
#define rtmGetStopRequested(rtm)       ((void*) 0)
#endif
#endif                                 /* RTW_HEADER_rtmodel_h_ */
```

#### rtwtypes.h
```c
/*
 * rtwtypes.h
 *
 * Academic License - for use in teaching, academic research, and meeting
 * course requirements at degree granting institutions only.  Not for
 * government, commercial, or other organizational use.
 *
 * Code generation for model "cyklovac_BB".
 *
 * Model version              : 1.8
 * Simulink Coder version : 9.6 (R2021b) 14-May-2021
 * C source code generated on : Thu Mar 17 07:18:42 2022
 *
 * Target selection: bur_grt.tlc
 * Note: GRT includes extra infrastructure and instrumentation for prototyping
 * Embedded hardware selection: Intel->x86/Pentium
 * Code generation objectives: Unspecified
 * Validation result: Not run
 */

#ifndef RTWTYPES_H
#define RTWTYPES_H
#include "tmwtypes.h"
#ifndef POINTER_T
#define POINTER_T

typedef void * pointer_T;

#endif

/* Logical type definitions */
#if (!defined(__cplusplus))
#ifndef false
#define false                          (0U)
#endif

#ifndef true
#define true                           (1U)
#endif
#endif
#endif                                 /* RTWTYPES_H */
```

### Library Logical/Libraries/regulatory (ANSIC, version 1.00.0)

#### reg_FF_PI_pl_regr_stiff.h
```c
/*
 * reg_FF_PI_pl_regr_stiff.h
 *
 * Academic License - for use in teaching, academic research, and meeting
 * course requirements at degree granting institutions only.  Not for
 * government, commercial, or other organizational use.
 *
 * Code generation for model "reg_FF_PI_pl_regr_stiff".
 *
 * Model version              : 1.135
 * Simulink Coder version : 9.6 (R2021b) 14-May-2021
 * C source code generated on : Tue Sep 27 10:51:43 2022
 *
 * Target selection: bur_grt.tlc
 * Note: GRT includes extra infrastructure and instrumentation for prototyping
 * Embedded hardware selection: Intel->x86/Pentium
 * Code generation objectives: Unspecified
 * Validation result: Not run
 */

#ifndef RTW_HEADER_reg_FF_PI_pl_regr_stiff_h_
#define RTW_HEADER_reg_FF_PI_pl_regr_stiff_h_
#include <math.h>
#include <stddef.h>
#include <string.h>
#ifndef reg_FF_PI_pl_regr_stiff_COMMON_INCLUDES_
#define reg_FF_PI_pl_regr_stiff_COMMON_INCLUDES_
#include <stdlib.h>
#include "rtwtypes.h"
#include "rtw_continuous.h"
#include "rtw_solver.h"
#endif                            /* reg_FF_PI_pl_regr_stiff_COMMON_INCLUDES_ */

#include "reg_FF_PI_pl_regr_stiff_types.h"
#include "regulatory.h"
/* Beginning of Dynamic TypeDefs: */
/* End of Dynamic TypeDefs: */
#ifndef MIN
#define MIN(a,b)	((a) < (b) ? (a) : (b))
#endif

#ifndef MAX
#define MAX(a,b)	((a) > (b) ? (a) : (b))
#endif

#ifndef AST_ROUND
#define AST_ROUND(x) ((x)>=0?(long long)((x)+0.5):(long long)((x)-0.5))
#endif

/* Shared type includes */
#include "multiword_types.h"

/* Macros for accessing real-time model data structure */
#ifndef rtmGetBlockIO
#define rtmGetBlockIO(rtm)             ((rtm)->blockIO)
#endif

#ifndef rtmSetBlockIO
#define rtmSetBlockIO(rtm, val)        ((rtm)->blockIO = (val))
#endif

#ifndef rtmGetRootDWork
#define rtmGetRootDWork(rtm)           ((rtm)->dwork)
#endif

#ifndef rtmSetRootDWork
#define rtmSetRootDWork(rtm, val)      ((rtm)->dwork = (val))
#endif

#ifndef rtmGetErrorStatus
#define rtmGetErrorStatus(rtm)         ((rtm)->errorStatus)
#endif

#ifndef rtmSetErrorStatus
#define rtmSetErrorStatus(rtm, val)    ((rtm)->errorStatus = (val))
#endif

#define reg_FF_PI_pl_regr_stiff_M_TYPE RT_MODEL_reg_FF_PI_pl_regr_st_T

/* Block signals (default storage) */

/* Block states (default storage) for system '<Root>' */

/* Constant parameters (default storage) */

/* Real-time Model Data Structure */

/* External data declarations for dependent source files */
extern const char *RT_MEMORY_ALLOCATION_ERROR;

/* Constant parameters (default storage) */
extern const ConstP_reg_FF_PI_pl_regr_stif_T reg_FF_PI_pl_regr_stiff_ConstP;

/* Model entry point functions */
extern void reg_FF_PI_pl_regr_stiff_initializeMemory(RT_MODEL_reg_FF_PI_pl_regr_st_T * const reg_FF_PI_pl_regr_stiff_M, struct FF_PID_r_t* inst);
extern void reg_FF_PI_pl_regr_stiff_initialize(RT_MODEL_reg_FF_PI_pl_regr_st_T *
  const reg_FF_PI_pl_regr_stiff_M, struct FF_PID_r_t* inst);
extern void reg_FF_PI_pl_regr_stiff_step(RT_MODEL_reg_FF_PI_pl_regr_st_T *const
  reg_FF_PI_pl_regr_stiff_M, struct FF_PID_r_t* inst);
extern void reg_FF_PI_pl_regr_stiff_terminate(RT_MODEL_reg_FF_PI_pl_regr_st_T
  * reg_FF_PI_pl_regr_stiff_M, struct FF_PID_r_t* inst);

/*-
 * The generated code includes comments that allow you to trace directly
 * back to the appropriate location in the model.  The basic format
 * is <system>/block_name, where system is the system number (uniquely
 * assigned by Simulink) and block_name is the name of the block.
 *
 * Use the MATLAB hilite_system command to trace the generated code back
 * to the model.  For example,
 *
 * hilite_system('<S3>')    - opens system 3
 * hilite_system('<S3>/Kp') - opens and selects block Kp which resides in S3
 *
 * Here is the system hierarchy for this model
 *
 * '<Root>' : 'reg_FF_PI_pl_regr_stiff'
 * '<S1>'   : 'reg_FF_PI_pl_regr_stiff/FF_zlozka'
 * '<S2>'   : 'reg_FF_PI_pl_regr_stiff/Subsystem'
 * '<S3>'   : 'reg_FF_PI_pl_regr_stiff/FF_zlozka/MATLAB Function'
 * '<S4>'   : 'reg_FF_PI_pl_regr_stiff/Subsystem/AlfaX_baseY2deltaz2'
 * '<S5>'   : 'reg_FF_PI_pl_regr_stiff/Subsystem/V_PID_Yellow'
 * '<S6>'   : 'reg_FF_PI_pl_regr_stiff/Subsystem/V_PID_Yellow1'
 * '<S7>'   : 'reg_FF_PI_pl_regr_stiff/Subsystem/V_PID_blue'
 * '<S8>'   : 'reg_FF_PI_pl_regr_stiff/Subsystem/abs2relat1'
 * '<S9>'   : 'reg_FF_PI_pl_regr_stiff/Subsystem/abs2relat2'
 * '<S10>'  : 'reg_FF_PI_pl_regr_stiff/Subsystem/abs2relat3'
 * '<S11>'  : 'reg_FF_PI_pl_regr_stiff/Subsystem/abs2relat4'
 * '<S12>'  : 'reg_FF_PI_pl_regr_stiff/Subsystem/abs2relat7'
 * '<S13>'  : 'reg_FF_PI_pl_regr_stiff/Subsystem/abs2relat8'
 * '<S14>'  : 'reg_FF_PI_pl_regr_stiff/Subsystem/AlfaX_baseY2deltaz2/requested alfa 2 deltaz1'
 * '<S15>'  : 'reg_FF_PI_pl_regr_stiff/Subsystem/V_PID_Yellow/Anti-windup'
 * '<S16>'  : 'reg_FF_PI_pl_regr_stiff/Subsystem/V_PID_Yellow/D Gain'
 * '<S17>'  : 'reg_FF_PI_pl_regr_stiff/Subsystem/V_PID_Yellow/Filter'
 * '<S18>'  : 'reg_FF_PI_pl_regr_stiff/Subsystem/V_PID_Yellow/Filter ICs'
 * '<S19>'  : 'reg_FF_PI_pl_regr_stiff/Subsystem/V_PID_Yellow/I Gain'
 * '<S20>'  : 'reg_FF_PI_pl_regr_stiff/Subsystem/V_PID_Yellow/Ideal P Gain'
 * '<S21>'  : 'reg_FF_PI_pl_regr_stiff/Subsystem/V_PID_Yellow/Ideal P Gain Fdbk'
 * '<S22>'  : 'reg_FF_PI_pl_regr_stiff/Subsystem/V_PID_Yellow/Integrator'
 * '<S23>'  : 'reg_FF_PI_pl_regr_stiff/Subsystem/V_PID_Yellow/Integrator ICs'
 * '<S24>'  : 'reg_FF_PI_pl_regr_stiff/Subsystem/V_PID_Yellow/N Copy'
 * '<S25>'  : 'reg_FF_PI_pl_regr_stiff/Subsystem/V_PID_Yellow/N Gain'
 * '<S26>'  : 'reg_FF_PI_pl_regr_stiff/Subsystem/V_PID_Yellow/P Copy'
 * '<S27>'  : 'reg_FF_PI_pl_regr_stiff/Subsystem/V_PID_Yellow/Parallel P Gain'
 * '<S28>'  : 'reg_FF_PI_pl_regr_stiff/Subsystem/V_PID_Yellow/Reset Signal'
 * '<S29>'  : 'reg_FF_PI_pl_regr_stiff/Subsystem/V_PID_Yellow/Saturation'
 * '<S30>'  : 'reg_FF_PI_pl_regr_stiff/Subsystem/V_PID_Yellow/Saturation Fdbk'
 * '<S31>'  : 'reg_FF_PI_pl_regr_stiff/Subsystem/V_PID_Yellow/Sum'
 * '<S32>'  : 'reg_FF_PI_pl_regr_stiff/Subsystem/V_PID_Yellow/Sum Fdbk'
 * '<S33>'  : 'reg_FF_PI_pl_regr_stiff/Subsystem/V_PID_Yellow/Tracking Mode'
 * '<S34>'  : 'reg_FF_PI_pl_regr_stiff/Subsystem/V_PID_Yellow/Tracking Mode Sum'
 * '<S35>'  : 'reg_FF_PI_pl_regr_stiff/Subsystem/V_PID_Yellow/Tsamp - Integral'
 * '<S36>'  : 'reg_FF_PI_pl_regr_stiff/Subsystem/V_PID_Yellow/Tsamp - Ngain'
 * '<S37>'  : 'reg_FF_PI_pl_regr_stiff/Subsystem/V_PID_Yellow/postSat Signal'
 * '<S38>'  : 'reg_FF_PI_pl_regr_stiff/Subsystem/V_PID_Yellow/preSat Signal'
 * '<S39>'  : 'reg_FF_PI_pl_regr_stiff/Subsystem/V_PID_Yellow/Anti-windup/Passthrough'
 * '<S40>'  : 'reg_FF_PI_pl_regr_stiff/Subsystem/V_PID_Yellow/D Gain/External Parameters'
 * '<S41>'  : 'reg_FF_PI_pl_regr_stiff/Subsystem/V_PID_Yellow/Filter/Disc. Forward Euler Filter'
 * '<S42>'  : 'reg_FF_PI_pl_regr_stiff/Subsystem/V_PID_Yellow/Filter ICs/Internal IC - Filter'
 * '<S43>'  : 'reg_FF_PI_pl_regr_stiff/Subsystem/V_PID_Yellow/I Gain/External Parameters'
 * '<S44>'  : 'reg_FF_PI_pl_regr_stiff/Subsystem/V_PID_Yellow/Ideal P Gain/Passthrough'
 * '<S45>'  : 'reg_FF_PI_pl_regr_stiff/Subsystem/V_PID_Yellow/Ideal P Gain Fdbk/Disabled'
 * '<S46>'  : 'reg_FF_PI_pl_regr_stiff/Subsystem/V_PID_Yellow/Integrator/Discrete'
 * '<S47>'  : 'reg_FF_PI_pl_regr_stiff/Subsystem/V_PID_Yellow/Integrator ICs/Internal IC'
 * '<S48>'  : 'reg_FF_PI_pl_regr_stiff/Subsystem/V_PID_Yellow/N Copy/Disabled'
 * '<S49>'  : 'reg_FF_PI_pl_regr_stiff/Subsystem/V_PID_Yellow/N Gain/External Parameters'
 * '<S50>'  : 'reg_FF_PI_pl_regr_stiff/Subsystem/V_PID_Yellow/P Copy/Disabled'
 * '<S51>'  : 'reg_FF_PI_pl_regr_stiff/Subsystem/V_PID_Yellow/Parallel P Gain/External Parameters'
 * '<S52>'  : 'reg_FF_PI_pl_regr_stiff/Subsystem/V_PID_Yellow/Reset Signal/External Reset'
 * '<S53>'  : 'reg_FF_PI_pl_regr_stiff/Subsystem/V_PID_Yellow/Saturation/External'
 * '<S54>'  : 'reg_FF_PI_pl_regr_stiff/Subsystem/V_PID_Yellow/Saturation/External/Saturation Dynamic'
 * '<S55>'  : 'reg_FF_PI_pl_regr_stiff/Subsystem/V_PID_Yellow/Saturation Fdbk/Disabled'
 * '<S56>'  : 'reg_FF_PI_pl_regr_stiff/Subsystem/V_PID_Yellow/Sum/Sum_PID'
 * '<S57>'  : 'reg_FF_PI_pl_regr_stiff/Subsystem/V_PID_Yellow/Sum Fdbk/Disabled'
 * '<S58>'  : 'reg_FF_PI_pl_regr_stiff/Subsystem/V_PID_Yellow/Tracking Mode/Disabled'
 * '<S59>'  : 'reg_FF_PI_pl_regr_stiff/Subsystem/V_PID_Yellow/Tracking Mode Sum/Passthrough'
 * '<S60>'  : 'reg_FF_PI_pl_regr_stiff/Subsystem/V_PID_Yellow/Tsamp - Integral/Passthrough'
 * '<S61>'  : 'reg_FF_PI_pl_regr_stiff/Subsystem/V_PID_Yellow/Tsamp - Ngain/Passthrough'
 * '<S62>'  : 'reg_FF_PI_pl_regr_stiff/Subsystem/V_PID_Yellow/postSat Signal/Forward_Path'
 * '<S63>'  : 'reg_FF_PI_pl_regr_stiff/Subsystem/V_PID_Yellow/preSat Signal/Forward_Path'
 * '<S64>'  : 'reg_FF_PI_pl_regr_stiff/Subsystem/V_PID_Yellow1/Anti-windup'
 * '<S65>'  : 'reg_FF_PI_pl_regr_stiff/Subsystem/V_PID_Yellow1/D Gain'
 * '<S66>'  : 'reg_FF_PI_pl_regr_stiff/Subsystem/V_PID_Yellow1/Filter'
 * '<S67>'  : 'reg_FF_PI_pl_regr_stiff/Subsystem/V_PID_Yellow1/Filter ICs'
 * '<S68>'  : 'reg_FF_PI_pl_regr_stiff/Subsystem/V_PID_Yellow1/I Gain'
 * '<S69>'  : 'reg_FF_PI_pl_regr_stiff/Subsystem/V_PID_Yellow1/Ideal P Gain'
 * '<S70>'  : 'reg_FF_PI_pl_regr_stiff/Subsystem/V_PID_Yellow1/Ideal P Gain Fdbk'
 * '<S71>'  : 'reg_FF_PI_pl_regr_stiff/Subsystem/V_PID_Yellow1/Integrator'
 * '<S72>'  : 'reg_FF_PI_pl_regr_stiff/Subsystem/V_PID_Yellow1/Integrator ICs'
 * '<S73>'  : 'reg_FF_PI_pl_regr_stiff/Subsystem/V_PID_Yellow1/N Copy'
 * '<S74>'  : 'reg_FF_PI_pl_regr_stiff/Subsystem/V_PID_Yellow1/N Gain'
 * '<S75>'  : 'reg_FF_PI_pl_regr_stiff/Subsystem/V_PID_Yellow1/P Copy'
 * '<S76>'  : 'reg_FF_PI_pl_regr_stiff/Subsystem/V_PID_Yellow1/Parallel P Gain'
 * '<S77>'  : 'reg_FF_PI_pl_regr_stiff/Subsystem/V_PID_Yellow1/Reset Signal'
 * '<S78>'  : 'reg_FF_PI_pl_regr_stiff/Subsystem/V_PID_Yellow1/Saturation'
 * '<S79>'  : 'reg_FF_PI_pl_regr_stiff/Subsystem/V_PID_Yellow1/Saturation Fdbk'
 * '<S80>'  : 'reg_FF_PI_pl_regr_stiff/Subsystem/V_PID_Yellow1/Sum'
 * '<S81>'  : 'reg_FF_PI_pl_regr_stiff/Subsystem/V_PID_Yellow1/Sum Fdbk'
 * '<S82>'  : 'reg_FF_PI_pl_regr_stiff/Subsystem/V_PID_Yellow1/Tracking Mode'
 * '<S83>'  : 'reg_FF_PI_pl_regr_stiff/Subsystem/V_PID_Yellow1/Tracking Mode Sum'
 * '<S84>'  : 'reg_FF_PI_pl_regr_stiff/Subsystem/V_PID_Yellow1/Tsamp - Integral'
 * '<S85>'  : 'reg_FF_PI_pl_regr_stiff/Subsystem/V_PID_Yellow1/Tsamp - Ngain'
 * '<S86>'  : 'reg_FF_PI_pl_regr_stiff/Subsystem/V_PID_Yellow1/postSat Signal'
 * '<S87>'  : 'reg_FF_PI_pl_regr_stiff/Subsystem/V_PID_Yellow1/preSat Signal'
 * '<S88>'  : 'reg_FF_PI_pl_regr_stiff/Subsystem/V_PID_Yellow1/Anti-windup/Passthrough'
 * '<S89>'  : 'reg_FF_PI_pl_regr_stiff/Subsystem/V_PID_Yellow1/D Gain/External Parameters'
 * '<S90>'  : 'reg_FF_PI_pl_regr_stiff/Subsystem/V_PID_Yellow1/Filter/Disc. Forward Euler Filter'
 * '<S91>'  : 'reg_FF_PI_pl_regr_stiff/Subsystem/V_PID_Yellow1/Filter ICs/Internal IC - Filter'
 * '<S92>'  : 'reg_FF_PI_pl_regr_stiff/Subsystem/V_PID_Yellow1/I Gain/External Parameters'
 * '<S93>'  : 'reg_FF_PI_pl_regr_stiff/Subsystem/V_PID_Yellow1/Ideal P Gain/Passthrough'
 * '<S94>'  : 'reg_FF_PI_pl_regr_stiff/Subsystem/V_PID_Yellow1/Ideal P Gain Fdbk/Disabled'
 * '<S95>'  : 'reg_FF_PI_pl_regr_stiff/Subsystem/V_PID_Yellow1/Integrator/Discrete'
 * '<S96>'  : 'reg_FF_PI_pl_regr_stiff/Subsystem/V_PID_Yellow1/Integrator ICs/Internal IC'
 * '<S97>'  : 'reg_FF_PI_pl_regr_stiff/Subsystem/V_PID_Yellow1/N Copy/Disabled'
 * '<S98>'  : 'reg_FF_PI_pl_regr_stiff/Subsystem/V_PID_Yellow1/N Gain/External Parameters'
 * '<S99>'  : 'reg_FF_PI_pl_regr_stiff/Subsystem/V_PID_Yellow1/P Copy/Disabled'
 * '<S100>' : 'reg_FF_PI_pl_regr_stiff/Subsystem/V_PID_Yellow1/Parallel P Gain/External Parameters'
 * '<S101>' : 'reg_FF_PI_pl_regr_stiff/Subsystem/V_PID_Yellow1/Reset Signal/External Reset'
 * '<S102>' : 'reg_FF_PI_pl_regr_stiff/Subsystem/V_PID_Yellow1/Saturation/External'
 * '<S103>' : 'reg_FF_PI_pl_regr_stiff/Subsystem/V_PID_Yellow1/Saturation/External/Saturation Dynamic'
 * '<S104>' : 'reg_FF_PI_pl_regr_stiff/Subsystem/V_PID_Yellow1/Saturation Fdbk/Disabled'
 * '<S105>' : 'reg_FF_PI_pl_regr_stiff/Subsystem/V_PID_Yellow1/Sum/Sum_PID'
 * '<S106>' : 'reg_FF_PI_pl_regr_stiff/Subsystem/V_PID_Yellow1/Sum Fdbk/Disabled'
 * '<S107>' : 'reg_FF_PI_pl_regr_stiff/Subsystem/V_PID_Yellow1/Tracking Mode/Disabled'
 * '<S108>' : 'reg_FF_PI_pl_regr_stiff/Subsystem/V_PID_Yellow1/Tracking Mode Sum/Passthrough'
 * '<S109>' : 'reg_FF_PI_pl_regr_stiff/Subsystem/V_PID_Yellow1/Tsamp - Integral/Passthrough'
 * '<S110>' : 'reg_FF_PI_pl_regr_stiff/Subsystem/V_PID_Yellow1/Tsamp - Ngain/Passthrough'
 * '<S111>' : 'reg_FF_PI_pl_regr_stiff/Subsystem/V_PID_Yellow1/postSat Signal/Forward_Path'
 * '<S112>' : 'reg_FF_PI_pl_regr_stiff/Subsystem/V_PID_Yellow1/preSat Signal/Forward_Path'
 * '<S113>' : 'reg_FF_PI_pl_regr_stiff/Subsystem/V_PID_blue/Anti-windup'
 * '<S114>' : 'reg_FF_PI_pl_regr_stiff/Subsystem/V_PID_blue/D Gain'
 * '<S115>' : 'reg_FF_PI_pl_regr_stiff/Subsystem/V_PID_blue/Filter'
 * '<S116>' : 'reg_FF_PI_pl_regr_stiff/Subsystem/V_PID_blue/Filter ICs'
 * '<S117>' : 'reg_FF_PI_pl_regr_stiff/Subsystem/V_PID_blue/I Gain'
 * '<S118>' : 'reg_FF_PI_pl_regr_stiff/Subsystem/V_PID_blue/Ideal P Gain'
 * '<S119>' : 'reg_FF_PI_pl_regr_stiff/Subsystem/V_PID_blue/Ideal P Gain Fdbk'
 * '<S120>' : 'reg_FF_PI_pl_regr_stiff/Subsystem/V_PID_blue/Integrator'
 * '<S121>' : 'reg_FF_PI_pl_regr_stiff/Subsystem/V_PID_blue/Integrator ICs'
 * '<S122>' : 'reg_FF_PI_pl_regr_stiff/Subsystem/V_PID_blue/N Copy'
 * '<S123>' : 'reg_FF_PI_pl_regr_stiff/Subsystem/V_PID_blue/N Gain'
 * '<S124>' : 'reg_FF_PI_pl_regr_stiff/Subsystem/V_PID_blue/P Copy'
 * '<S125>' : 'reg_FF_PI_pl_regr_stiff/Subsystem/V_PID_blue/Parallel P Gain'
 * '<S126>' : 'reg_FF_PI_pl_regr_stiff/Subsystem/V_PID_blue/Reset Signal'
 * '<S127>' : 'reg_FF_PI_pl_regr_stiff/Subsystem/V_PID_blue/Saturation'
 * '<S128>' : 'reg_FF_PI_pl_regr_stiff/Subsystem/V_PID_blue/Saturation Fdbk'
 * '<S129>' : 'reg_FF_PI_pl_regr_stiff/Subsystem/V_PID_blue/Sum'
 * '<S130>' : 'reg_FF_PI_pl_regr_stiff/Subsystem/V_PID_blue/Sum Fdbk'
 * '<S131>' : 'reg_FF_PI_pl_regr_stiff/Subsystem/V_PID_blue/Tracking Mode'
 * '<S132>' : 'reg_FF_PI_pl_regr_stiff/Subsystem/V_PID_blue/Tracking Mode Sum'
 * '<S133>' : 'reg_FF_PI_pl_regr_stiff/Subsystem/V_PID_blue/Tsamp - Integral'
 * '<S134>' : 'reg_FF_PI_pl_regr_stiff/Subsystem/V_PID_blue/Tsamp - Ngain'
 * '<S135>' : 'reg_FF_PI_pl_regr_stiff/Subsystem/V_PID_blue/postSat Signal'
 * '<S136>' : 'reg_FF_PI_pl_regr_stiff/Subsystem/V_PID_blue/preSat Signal'
 * '<S137>' : 'reg_FF_PI_pl_regr_stiff/Subsystem/V_PID_blue/Anti-windup/Passthrough'
 * '<S138>' : 'reg_FF_PI_pl_regr_stiff/Subsystem/V_PID_blue/D Gain/External Parameters'
 * '<S139>' : 'reg_FF_PI_pl_regr_stiff/Subsystem/V_PID_blue/Filter/Disc. Forward Euler Filter'
 * '<S140>' : 'reg_FF_PI_pl_regr_stiff/Subsystem/V_PID_blue/Filter ICs/Internal IC - Filter'
 * '<S141>' : 'reg_FF_PI_pl_regr_stiff/Subsystem/V_PID_blue/I Gain/External Parameters'
 * '<S142>' : 'reg_FF_PI_pl_regr_stiff/Subsystem/V_PID_blue/Ideal P Gain/Passthrough'
 * '<S143>' : 'reg_FF_PI_pl_regr_stiff/Subsystem/V_PID_blue/Ideal P Gain Fdbk/Disabled'
 * '<S144>' : 'reg_FF_PI_pl_regr_stiff/Subsystem/V_PID_blue/Integrator/Discrete'
 * '<S145>' : 'reg_FF_PI_pl_regr_stiff/Subsystem/V_PID_blue/Integrator ICs/Internal IC'
 * '<S146>' : 'reg_FF_PI_pl_regr_stiff/Subsystem/V_PID_blue/N Copy/Disabled'
 * '<S147>' : 'reg_FF_PI_pl_regr_stiff/Subsystem/V_PID_blue/N Gain/External Parameters'
 * '<S148>' : 'reg_FF_PI_pl_regr_stiff/Subsystem/V_PID_blue/P Copy/Disabled'
 * '<S149>' : 'reg_FF_PI_pl_regr_stiff/Subsystem/V_PID_blue/Parallel P Gain/External Parameters'
 * '<S150>' : 'reg_FF_PI_pl_regr_stiff/Subsystem/V_PID_blue/Reset Signal/External Reset'
 * '<S151>' : 'reg_FF_PI_pl_regr_stiff/Subsystem/V_PID_blue/Saturation/External'
 * '<S152>' : 'reg_FF_PI_pl_regr_stiff/Subsystem/V_PID_blue/Saturation/External/Saturation Dynamic'
 * '<S153>' : 'reg_FF_PI_pl_regr_stiff/Subsystem/V_PID_blue/Saturation Fdbk/Disabled'
 * '<S154>' : 'reg_FF_PI_pl_regr_stiff/Subsystem/V_PID_blue/Sum/Sum_PID'
 * '<S155>' : 'reg_FF_PI_pl_regr_stiff/Subsystem/V_PID_blue/Sum Fdbk/Disabled'
 * '<S156>' : 'reg_FF_PI_pl_regr_stiff/Subsystem/V_PID_blue/Tracking Mode/Disabled'
 * '<S157>' : 'reg_FF_PI_pl_regr_stiff/Subsystem/V_PID_blue/Tracking Mode Sum/Passthrough'
 * '<S158>' : 'reg_FF_PI_pl_regr_stiff/Subsystem/V_PID_blue/Tsamp - Integral/Passthrough'
 * '<S159>' : 'reg_FF_PI_pl_regr_stiff/Subsystem/V_PID_blue/Tsamp - Ngain/Passthrough'
 * '<S160>' : 'reg_FF_PI_pl_regr_stiff/Subsystem/V_PID_blue/postSat Signal/Forward_Path'
 * '<S161>' : 'reg_FF_PI_pl_regr_stiff/Subsystem/V_PID_blue/preSat Signal/Forward_Path'
 */
#endif                               /* RTW_HEADER_reg_FF_PI_pl_regr_stiff_h_ */
```

#### reg_FF_PI_pl_regr_stiff_data.c
```c
/*
 * reg_FF_PI_pl_regr_stiff_data.c
 *
 * Academic License - for use in teaching, academic research, and meeting
 * course requirements at degree granting institutions only.  Not for
 * government, commercial, or other organizational use.
 *
 * Code generation for model "reg_FF_PI_pl_regr_stiff".
 *
 * Model version              : 1.135
 * Simulink Coder version : 9.6 (R2021b) 14-May-2021
 * C source code generated on : Tue Sep 27 10:51:43 2022
 *
 * Target selection: bur_grt.tlc
 * Note: GRT includes extra infrastructure and instrumentation for prototyping
 * Embedded hardware selection: Intel->x86/Pentium
 * Code generation objectives: Unspecified
 * Validation result: Not run
 */

#include "reg_FF_PI_pl_regr_stiff.h"
#include "reg_FF_PI_pl_regr_stiff_private.h"

/* Constant parameters (default storage) */
const ConstP_reg_FF_PI_pl_regr_stif_T reg_FF_PI_pl_regr_stiff_ConstP = {
  /* Expression: coef_1blue
   * Referenced by: '<S1>/Constant'
   */
  { 0.0017105750782315647, -0.00031894042792665118, 0.00035451787790138196,
    -0.00019972200976834959, -4.3892191255761959E-6, -0.00027272249934474538,
    -0.0090478565722579233, 0.0054482716433918608, -0.0072683292922697922,
    0.00413929721958372, 0.00011303098682474825, 0.005591677047672953,
    -0.16681175073563032, -0.036143207245384182, 0.061165365811016628,
    -0.035360608238866748, -0.0011446751359908019, -0.047290107610719861,
    1.9314414355397496, 0.11599151682470536, -0.27274287157744381,
    0.16106157257347073, 0.0059214601396658942, 0.21348955813855988,
    -8.214194337602315, -0.17468404062406745, 0.6935075165131781,
    -0.42202772508074771, -0.016877335878941583, -0.55515365502246838,
    17.123747629688115, 0.0669008896991383, -1.0026784691064161,
    0.63585828567519109, 0.026421042370275552, 0.831151470907112,
    -16.462934654986736, 0.079274206258717048, 0.76227189768315973,
    -0.50974126037567646, -0.020778480585300123, -0.66377130446245836,
    6.95932519589881, -0.12150704958189475, -0.2350544296785472,
    0.16808162279516273, 0.0063626246901319922, 0.21805719235011847 },

  /* Expression: coef_2green
   * Referenced by: '<S1>/Constant1'
   */
  { -0.00038837768098208894, -0.00065117847140775634, 0.00020964331658933648,
    -0.00018966178503272696, 3.6107136311502476E-5, -0.00024567775366209614,
    0.040858546502079623, 0.013145297264238857, -0.0038628601851493733,
    0.00381104087840559, -0.00078121720792697876, 0.00494457781501693,
    -0.65271977929603131, -0.10904154399504047, 0.029139742826547764,
    -0.031407923824548177, 0.007065116461826647, -0.040866436032779611,
    4.4274857655001005, 0.48099251537940674, -0.11739905582318358,
    0.13731679994241536, -0.034458101183743185, 0.17944913231215021,
    -15.481147119163195, -1.2192478431872231, 0.27498378684430841,
    -0.3438802890129693, 0.0971390050296614, -0.45202364142946455,
    29.093533123706937, 1.7796492959360444, -0.37826210079672062,
    0.49388247912156341, -0.15713393344808899, 0.65356045383838535,
    -26.820653555856456, -1.3767944130597296, 0.30889409220045694,
    -0.37750822598435141, 0.13499544127719082, -0.50254981985427571,
    10.589080614584185, 0.46805035762142011, -0.055008004115544067,
    0.11889561406308008, -0.048021210874138291, 0.15896689069549794 },

  /* Expression: coef_3yellow
   * Referenced by: '<S1>/Constant3'
   */
  { 0.0040655521860770679, -0.00045625459374585214, 0.00039587384671225151,
    -0.00028172651766770795, -6.7214130921795348E-5, -0.00028248251395603281,
    -0.052274548967079511, 0.0084304027358908049, -0.0084374664797956141,
    0.0058331765704457876, 0.0015123649012436069, 0.0056840040026990453,
    0.15271371298337824, -0.062075974257985153, 0.073622574381782768,
    -0.049821467704821772, -0.014136189017056839, -0.0469477448909448,
    0.70330100029796949, 0.2325052510651455, -0.33964790581471743,
    0.22704315289173943, 0.070767737933930264, 0.20592112565908618,
    -5.5665529664061006, -0.46853556022720089, 0.89425321396155255,
    -0.59536150815747069, -0.20361499567782843, -0.51788809106330591,
    13.92427212519536, 0.487773373707155, -1.3442475203161097,
    0.89740396531665878, 0.33491638476311841, 0.7474525928110074,
    -14.331234712148808, -0.20455292310497739, 1.0456791951890665,
    -0.71989856223038, -0.29138519106015026, -0.57384727370638533,
    6.25235418888368, 0.032212696269155724, -0.38388460202577607,
    0.23671769120847469, 0.10374886423005664, 0.18103901615539519 }
};
```

#### reg_FF_PI_pl_regr_stiff_private.h
```c
/*
 * reg_FF_PI_pl_regr_stiff_private.h
 *
 * Academic License - for use in teaching, academic research, and meeting
 * course requirements at degree granting institutions only.  Not for
 * government, commercial, or other organizational use.
 *
 * Code generation for model "reg_FF_PI_pl_regr_stiff".
 *
 * Model version              : 1.135
 * Simulink Coder version : 9.6 (R2021b) 14-May-2021
 * C source code generated on : Tue Sep 27 10:51:43 2022
 *
 * Target selection: bur_grt.tlc
 * Note: GRT includes extra infrastructure and instrumentation for prototyping
 * Embedded hardware selection: Intel->x86/Pentium
 * Code generation objectives: Unspecified
 * Validation result: Not run
 */

#ifndef RTW_HEADER_reg_FF_PI_pl_regr_stiff_private_h_
#define RTW_HEADER_reg_FF_PI_pl_regr_stiff_private_h_
#include "rtwtypes.h"
#include "multiword_types.h"
#if !defined(rt_VALIDATE_MEMORY)
#define rt_VALIDATE_MEMORY(S, ptr)     if(!(ptr)) {\
 rtmSetErrorStatus(reg_FF_PI_pl_regr_stiff_M, RT_MEMORY_ALLOCATION_ERROR);\
 }
#endif

#if !defined(rt_FREE)
#if !defined(_WIN32)
#define rt_FREE(ptr)                   if((ptr) != (NULL)) {\
 free((ptr));\
 (ptr) = (NULL);\
 }
#else

/* Visual and other windows compilers declare free without const */
#define rt_FREE(ptr)                   if((ptr) != (NULL)) {\
 free((void *)(ptr));\
 (ptr) = (NULL);\
 }
#endif
#endif
#endif                       /* RTW_HEADER_reg_FF_PI_pl_regr_stiff_private_h_ */
```

#### reg_FF_PI_pl_regr_stiff_types.h
```c
/*
 * reg_FF_PI_pl_regr_stiff_types.h
 *
 * Academic License - for use in teaching, academic research, and meeting
 * course requirements at degree granting institutions only.  Not for
 * government, commercial, or other organizational use.
 *
 * Code generation for model "reg_FF_PI_pl_regr_stiff".
 *
 * Model version              : 1.135
 * Simulink Coder version : 9.6 (R2021b) 14-May-2021
 * C source code generated on : Tue Sep 27 10:51:43 2022
 *
 * Target selection: bur_grt.tlc
 * Note: GRT includes extra infrastructure and instrumentation for prototyping
 * Embedded hardware selection: Intel->x86/Pentium
 * Code generation objectives: Unspecified
 * Validation result: Not run
 */

#ifndef RTW_HEADER_reg_FF_PI_pl_regr_stiff_types_h_
#define RTW_HEADER_reg_FF_PI_pl_regr_stiff_types_h_

/* Model Code Variants */

/* Forward declaration for rtModel */

#endif                         /* RTW_HEADER_reg_FF_PI_pl_regr_stiff_types_h_ */
```

#### regulatory.typ
```iecst
TYPE
	emxArray_real_T :  STRUCT
		data :  REFERENCE TO LREAL;
		size :  REFERENCE TO DINT;
		allocatedSize :  DINT;
		numDimensions :  DINT;
		canFreeData :  BOOL;
	END_STRUCT;

	B_regulator_FF_PI_T :  STRUCT
		Input1 :  REAL;
		Input2 :  REAL;
		Input3 :  REAL;
		Input4 :  REAL;
		Input11 :  REAL;
		Input5 :  REAL;
		Input13 :  REAL;
		Input14 :  REAL;
		Input8 :  REAL;
		Input9 :  REAL;
		Input10 :  REAL;
		Sum :  REAL;
		Input7 :  REAL;
		Sum2 :  REAL;
		Input6 :  REAL;
		Sum1 :  REAL;
		Input12 :  REAL;
	END_STRUCT;

	DW_regulator_FF_PI_T :  STRUCT
		Integrator_DSTATE :  LREAL;
		Filter_DSTATE :  LREAL;
		Integrator_DSTATE_o :  LREAL;
		Filter_DSTATE_f :  LREAL;
		Integrator_DSTATE_i :  LREAL;
		Filter_DSTATE_a :  LREAL;
		Integrator_PrevResetState :  SINT;
		Filter_PrevResetState :  SINT;
		Integrator_PrevResetState_l :  SINT;
		Filter_PrevResetState_e :  SINT;
		Integrator_PrevResetState_e :  SINT;
		Filter_PrevResetState_h :  SINT;
	END_STRUCT;

	ConstP_regulator_FF_PI_T :  STRUCT
		Constant_Value_m :  ARRAY[0..113] OF REAL;
		Constant1_Value_b :  ARRAY[0..113] OF REAL;
		Constant2_Value :  ARRAY[0..113] OF REAL;
		Constant3_Value :  ARRAY[0..113] OF REAL;
	END_STRUCT;

	tag_RTM_regulator_FF_PI_T :  STRUCT
		errorStatus :  REFERENCE TO USINT;
		blockIO :  REFERENCE TO B_regulator_FF_PI_T;
		dwork :  REFERENCE TO DW_regulator_FF_PI_T;
	END_STRUCT;

	B_regulator_FF_PI_plane_regre_T :  STRUCT
		Input1 :  REAL;
		Input2 :  REAL;
		Input3 :  REAL;
		Input4 :  REAL;
		Input11 :  REAL;
		Input5 :  REAL;
		Input13 :  REAL;
		Input14 :  REAL;
		Sum :  REAL;
		Input7 :  REAL;
		Sum2 :  REAL;
		Input6 :  REAL;
		Sum1 :  REAL;
		Input10 :  REAL;
		Input12 :  REAL;
		Input8 :  REAL;
		Input9 :  REAL;
	END_STRUCT;

	DW_regulator_FF_PI_plane_regr_T :  STRUCT
		Integrator_DSTATE :  LREAL;
		Filter_DSTATE :  LREAL;
		Integrator_DSTATE_o :  LREAL;
		Filter_DSTATE_f :  LREAL;
		Integrator_DSTATE_i :  LREAL;
		Filter_DSTATE_a :  LREAL;
		Integrator_PrevResetState :  SINT;
		Filter_PrevResetState :  SINT;
		Integrator_PrevResetState_l :  SINT;
		Filter_PrevResetState_e :  SINT;
		Integrator_PrevResetState_e :  SINT;
		Filter_PrevResetState_h :  SINT;
	END_STRUCT;

	tag_RTM_regulator_FF_PI_plane_T :  STRUCT
		errorStatus :  REFERENCE TO USINT;
		blockIO :  REFERENCE TO B_regulator_FF_PI_plane_regre_T;
		dwork :  REFERENCE TO DW_regulator_FF_PI_plane_regr_T;
	END_STRUCT;

	B_PID_constant_T :  STRUCT
		Input1 :  REAL;
		Input2 :  REAL;
		Input3 :  REAL;
		Input4 :  REAL;
		Input11 :  REAL;
		Input5 :  REAL;
		Input13 :  REAL;
		Input14 :  REAL;
		Switch2 :  REAL;
		Input6 :  REAL;
		Switch1 :  REAL;
		Input7 :  REAL;
		Switch :  REAL;
		Input12 :  REAL;
	END_STRUCT;

	DW_PID_constant_T :  STRUCT
		Integrator_DSTATE :  LREAL;
		Filter_DSTATE :  LREAL;
		Integrator_DSTATE_f :  LREAL;
		Filter_DSTATE_j :  LREAL;
		Integrator_DSTATE_h :  LREAL;
		Filter_DSTATE_m :  LREAL;
		Integrator_PrevResetState :  SINT;
		Filter_PrevResetState :  SINT;
		Integrator_PrevResetState_m :  SINT;
		Filter_PrevResetState_e :  SINT;
		Integrator_PrevResetState_l :  SINT;
		Filter_PrevResetState_k :  SINT;
	END_STRUCT;

	tag_RTM_PID_constant_T :  STRUCT
		errorStatus :  REFERENCE TO USINT;
		blockIO :  REFERENCE TO B_PID_constant_T;
		dwork :  REFERENCE TO DW_PID_constant_T;
	END_STRUCT;

	B_requestedalfa2deltaz1_reg_F_T :  STRUCT
		Blue_real :  REAL;
		Green_real :  REAL;
		Yellow_real :  REAL;
		Blue_ref :  REAL;
		Green_ref :  REAL;
		Yellow_ref :  REAL;
	END_STRUCT;

	B_regulator_nelin_P_T :  STRUCT
		Input1 :  REAL;
		Input2 :  REAL;
		Input3 :  REAL;
		Input4 :  REAL;
		Gain7 :  REAL;
		Gain9 :  REAL;
		Gain8 :  REAL;
	END_STRUCT;

	tag_RTM_regulator_nelin_P_T :  STRUCT
		errorStatus :  REFERENCE TO USINT;
		blockIO :  REFERENCE TO B_regulator_nelin_P_T;
	END_STRUCT;

	B_PID_co_T :  STRUCT
		Input1 :  REAL;
		Input2 :  REAL;
		Input3 :  REAL;
		Input4 :  REAL;
		Input11 :  REAL;
		Input5 :  REAL;
		Input13 :  REAL;
		Input14 :  REAL;
		Switch2 :  REAL;
		Input6 :  REAL;
		Switch1 :  REAL;
		Input7 :  REAL;
		Switch :  REAL;
		Input12 :  REAL;
	END_STRUCT;

	DW_PID_co_T :  STRUCT
		Integrator_DSTATE :  LREAL;
		Filter_DSTATE :  LREAL;
		Integrator_DSTATE_f :  LREAL;
		Filter_DSTATE_j :  LREAL;
		Integrator_DSTATE_h :  LREAL;
		Filter_DSTATE_m :  LREAL;
		Integrator_PrevResetState :  SINT;
		Filter_PrevResetState :  SINT;
		Integrator_PrevResetState_m :  SINT;
		Filter_PrevResetState_e :  SINT;
		Integrator_PrevResetState_l :  SINT;
		Filter_PrevResetState_k :  SINT;
	END_STRUCT;

	tag_RTM_PID_co_T :  STRUCT
		errorStatus :  REFERENCE TO USINT;
		blockIO :  REFERENCE TO B_PID_co_T;
		dwork :  REFERENCE TO DW_PID_co_T;
	END_STRUCT;

	B_reg_FF_PI_pl_regr_stiff_T :  STRUCT
		Input15 :  REAL;
		Input1 :  REAL;
		Input2 :  REAL;
		Input3 :  REAL;
		Input4 :  REAL;
		Input11 :  REAL;
		Input5 :  REAL;
		Input13 :  REAL;
		Input14 :  REAL;
		Sum :  REAL;
		Input7 :  REAL;
		Sum2 :  REAL;
		Input6 :  REAL;
		Sum1 :  REAL;
		Input10 :  REAL;
		Input12 :  REAL;
		Input8 :  REAL;
		Input9 :  REAL;
	END_STRUCT;

	DW_reg_FF_PI_pl_regr_stiff_T :  STRUCT
		Integrator_DSTATE :  LREAL;
		Filter_DSTATE :  LREAL;
		Integrator_DSTATE_o :  LREAL;
		Filter_DSTATE_f :  LREAL;
		Integrator_DSTATE_i :  LREAL;
		Filter_DSTATE_a :  LREAL;
		Integrator_PrevResetState :  SINT;
		Filter_PrevResetState :  SINT;
		Integrator_PrevResetState_l :  SINT;
		Filter_PrevResetState_e :  SINT;
		Integrator_PrevResetState_e :  SINT;
		Filter_PrevResetState_h :  SINT;
	END_STRUCT;

	ConstP_reg_FF_PI_pl_regr_stif_T :  STRUCT
		Constant_Value :  ARRAY[0..47] OF LREAL;
		Constant1_Value :  ARRAY[0..47] OF LREAL;
		Constant3_Value :  ARRAY[0..47] OF LREAL;
	END_STRUCT;

	tag_RTM_reg_FF_PI_pl_regr_sti_T :  STRUCT
		errorStatus :  REFERENCE TO USINT;
		blockIO :  REFERENCE TO B_reg_FF_PI_pl_regr_stiff_T;
		dwork :  REFERENCE TO DW_reg_FF_PI_pl_regr_stiff_T;
	END_STRUCT;

	emxArray_real_T_regulator_FF_T2 :emxArray_real_T;	(*  *)

	RT_MODEL_regulator_FF_PI_T :tag_RTM_regulator_FF_PI_T;	(*  *)

	RT_MODEL_regulator_FF_PI_plan_T :tag_RTM_regulator_FF_PI_plane_T;	(*  *)

	RT_MODEL_PID_constant_T :tag_RTM_PID_constant_T;	(*  *)

	RT_MODEL_regulator_nelin_P_T :tag_RTM_regulator_nelin_P_T;	(*  *)

	RT_MODEL_PID_co_T :tag_RTM_PID_co_T;	(*  *)

	RT_MODEL_reg_FF_PI_pl_regr_st_T :tag_RTM_reg_FF_PI_pl_regr_sti_T;	(*  *)

END_TYPE
```

### Program Logical/Source/Program (IEC)

#### Cyclic.st
```iecst
PROGRAM _CYCLIC

	IF tlacidla.zapni=TRUE THEN

		FOR i:=0 TO 7 BY 1 DO
			regulatory.reg[i] := REAL_TO_INT(display.in_reg[i]/100*32765/9);
		END_FOR

	ELSE

		FOR i:=0 TO 3 BY 1 DO
			tlacidla.ventil[i] := FALSE;
		END_FOR

		FOR i:=0 TO 7 BY 1 DO
			regulatory.reg[i] := 0;
		END_FOR

	END_IF

END_PROGRAM
```

#### Init.st
```iecst
PROGRAM _INIT
	(* Insert code here *)

END_PROGRAM
```

### LibAsUDP1_ST.typ
```iecst
(********************************************************************
 * COPYRIGHT -- Bernecker + Rainer
 ********************************************************************
 * File: Global.typ
 * Author: Bernecker + Rainer
 * Created: June 02, 2008
 ********************************************************************
 * Global data types of project LibAsUDP
 ********************************************************************)

TYPE
	LibAsUDP1_ST_typ : 	STRUCT  (*Datatyp for global Variables*)
		receive_data : ARRAY[0..100] OF UDINT; (*Data which has been received*)
		send_data : ARRAY[0..100] OF UDINT; (*Data which should be sent*)
	END_STRUCT;
END_TYPE
```

### Program Logical/Source/UDP/Client

#### Client.st
```iecst
(********************************************************************
 * COPYRIGHT -- Bernecker + Rainer
 ********************************************************************
 * Program: Client
 * File: Client.st
 * Author: Bernecker + Rainer
 * Created: June 02, 2008
 ********************************************************************
 * Implementation of program Client
 ********************************************************************)

PROGRAM _CYCLIC

	LibAsUDP1_ST.send_data[0] := LibAsUDP1_ST.send_data[0] + 1;  (* Generate a "running" variable for Data transfer *)

	CASE Client.sStep OF

		0:	(* Open UDP Port *)
			Client.UdpOpen_0.enable := 1;
			Client.UdpOpen_0.pIfAddr := 0;	(* Listen on all TCP/IP Interfaces*)
			Client.UdpOpen_0.port := 12051;	(* Port to listen*)
			Client.UdpOpen_0.options := 0;
			Client.UdpOpen_0;	(* Call the Function*)

			IF Client.UdpOpen_0.status = 0 THEN  (* UdpOpen successful*)
				Client.sStep := 1;
			ELSIF Client.UdpOpen_0.status = ERR_FUB_BUSY THEN  (* UdpOpen not finished -> redo *)
			  (* Busy *)
			ELSE  (* Goto Error Step *)
				Client.sStep := 10;
			END_IF

		1:	(* Send Data to the Server *)
			Client.server_address := '192.168.1.506';	(* IP Address of the Server *)
			Client.server_portnumber := 12050;	(* Port number of the Server *)

			Client.UdpSend_0.enable := 1;
			Client.UdpSend_0.ident := Client.UdpOpen_0.ident;	(* Connection Ident from AsUDP.UDP_Open *)
			Client.UdpSend_0.pHost := ADR(Client.server_address);
			Client.UdpSend_0.port := Client.server_portnumber;
			Client.UdpSend_0.pData := ADR(LibAsUDP1_ST.send_data);	(* Which data to send *)
			Client.UdpSend_0.datalen := SIZEOF(LibAsUDP1_ST.send_data);	(* Lenght of data to send *)
			Client.UdpSend_0.flags := 0;
			Client.UdpSend_0;	(* Call the Function*)

			IF Client.UdpSend_0.status = 0 THEN  (* Data sent *)
				Client.sStep := 2;
			ELSIF Client.UdpSend_0.status = ERR_FUB_BUSY THEN  (* UdpSend not finished -> redo *)
			  (* Busy *)
			ELSE  (* Goto Error Step *)
				Client.sStep := 10;
			END_IF

		2:	(* Receive Data from the Server *)
			Client.UdpRecv_0.enable := 1;
			Client.UdpRecv_0.ident := Client.UdpOpen_0.ident;  (* Connection Ident from AsUDP.UDP_Open *)
			Client.UdpRecv_0.pData	:= ADR(LibAsUDP1_ST.receive_data);  (* Where to store the incoming data *)
			Client.UdpRecv_0.datamax := SIZEOF(LibAsUDP1_ST.receive_data);  (* Lenght of data buffer *)
			Client.UdpRecv_0.flags := 0;
			Client.UdpRecv_0;  (* Call the Function*)

			IF Client.UdpRecv_0.status = 0 THEN  (* Data was received successfully -> Send next packet *)
				Client.sStep := 3;
				Client.no_data_received_count := 0;
			ELSIF Client.UdpRecv_0.status = udpERR_NO_DATA THEN  (* No data received - wait *)
			  (* No Data received *)
			  	Client.no_data_received_count := Client.no_data_received_count + 1;	(* Increase if no data are received *)

				IF Client.no_data_received_count > 200 THEN		(* No data timeout for TC1 [10ms] *)
					Client.no_data_received_count := 0;
					Client.sStep := 1;	(* Send again *)
				END_IF
			ELSIF Client.UdpRecv_0.status = ERR_FUB_BUSY THEN  (* UdpRecv not finished -> redo *)
			  (* Busy *)
			ELSE  (* Goto Error Step *)
				Client.sStep := 10;
			END_IF

		3: (* Close connection *)
			Client.UdpClose_0.enable := 1;
			Client.UdpClose_0.ident := Client.UdpOpen_0.ident;  (* Connection Ident from AsUDP.UDP_Open *)
			Client.UdpClose_0;  (* Call the Function*)

			IF Client.UdpClose_0.status = 0 THEN  (* Close successful -> Reopen the interface *)
				Client.sStep := 0;
			ELSIF Client.UdpClose_0.status = ERR_FUB_BUSY THEN  (* UdpClose not finished -> redo *)
			  (* Busy *)
			ELSE  (* Goto Error Step *)
				Client.sStep := 10;
			END_IF

		10: (* Here some error Handling has to be implemented *)

	END_CASE

END_PROGRAM
```

### Program Logical/Source/UDP/Server

#### Server.typ
```iecst
(********************************************************************
 * COPYRIGHT -- Bernecker + Rainer
 ********************************************************************
 * Program: Server
 * File: Server.typ
 * Author: Bernecker + Rainer
 * Created: June 02, 2008
 ********************************************************************
 * Local data types of program Server
 ********************************************************************)

TYPE
	Server_typ : 	STRUCT  (*UDP Server Variables*)
		sStep : UINT; (*UDP Server Step Variable*)
		client_address : STRING[20]; (*Address of the client connection to the Server*)
		UdpOpen_0 : UdpOpen; (*AsUDP.UdpOpen FUB*)
		UdpConnect_0 : UdpConnect; (*AsUDP.UdpConnect FUB*)
		UdpSend_0 : UdpSend; (*AsUDP.UdpSend FUB*)
		UdpRecv_0 : UdpRecv; (*AsUDP.UdpRecv FUB*)
		UdpDisconnect_0 : UdpDisconnect; (*AsUDP.UdpDisconnect FUB*)
		UdpClose_0 : UdpClose; (*AsUDP.UdpClose FUB*)
		data_buffer : ARRAY[0..100] OF UDINT; (*Data buffer ( receive and send )*)
	END_STRUCT;
END_TYPE
```

#### Server.var
```iecst
(********************************************************************
 * COPYRIGHT -- Bernecker + Rainer
 ********************************************************************
 * Program: Server
 * File: Server.var
 * Author: Bernecker + Rainer
 * Created: June 02, 2008
 ********************************************************************
 * Local variables of program Server
 ********************************************************************)
VAR
	Server : Server_typ := (0); (*Data for Server Task*)
	i : INT;
END_VAR
```

#### Server.st
```iecst
(********************************************************************
 * COPYRIGHT -- Bernecker + Rainer
 ********************************************************************
 * Program: Server
 * File: Server.st
 * Author: Bernecker + Rainer
 * Created: June 02, 2008
 ********************************************************************
 * Implementation of program Server
 ********************************************************************)

PROGRAM _CYCLIC

	// Receiving data from PC
	IF tlacidla.zapni = TRUE THEN

		CASE Server.sStep OF

			0:	(* Open UDP Port *)
				Server.UdpOpen_0.enable := 1;
				Server.UdpOpen_0.pIfAddr := 0;	(* Listen on all TCP/IP Interfaces*)
				Server.UdpOpen_0.port := 12050;	(* Port to listen*)
				Server.UdpOpen_0.options := 0;
				Server.UdpOpen_0;	(* Call the Function*)

				IF Server.UdpOpen_0.status = 0 THEN  (* UdpOpen successful*)
					Server.sStep := 1;
				ELSIF Server.UdpOpen_0.status = ERR_FUB_BUSY THEN  (* UdpOpen not finished -> redo *)
				  (* Busy *)
				ELSE  (* Goto Error Step *)
					Server.sStep := 10;
				END_IF

			1:	(* Wait for Data *)
				Server.UdpRecv_0.enable := 1;
				Server.UdpRecv_0.ident := Server.UdpOpen_0.ident;	(* Client Ident from AsUDP.UDP_Open *)
				Server.UdpRecv_0.pData := ADR(Server.data_buffer);	(* Where to store the incoming data *)
				Server.UdpRecv_0.datamax := SIZEOF(Server.data_buffer);	(* Lenght of data buffer *)
				Server.UdpRecv_0.flags := 0;
				Server.UdpRecv_0.pIpAddr := ADR(Server.client_address);	(* IP Address of the Client *)
				Server.UdpRecv_0;	(* Call the Function*)

				IF Server.UdpRecv_0.status = 0 THEN  (* Data received *)
					Server.sStep := 2;
				ELSIF Server.UdpRecv_0.status = udpERR_NO_DATA THEN  (* No data received - wait *)
				  (* No Data received *)
				ELSIF Server.UdpRecv_0.status = ERR_FUB_BUSY THEN  (* UdpRecv not finished -> redo *)
				  (* Busy *)
				ELSE  (* Goto Error Step *)
					Server.sStep := 10;
				END_IF

			2:	(* Send Data back to Client *)
				Server.UdpSend_0.enable := 1;
				Server.UdpSend_0.ident := Server.UdpOpen_0.ident;	(* Client Ident from AsUDP.UDP_Open *)
				Server.UdpSend_0.pHost := ADR(Server.client_address);	(* IP Address of the Client *)
				Server.UdpSend_0.port := Server.UdpRecv_0.port;		(* Port number of the Client *)
				Server.UdpSend_0.pData := ADR(Server.data_buffer);	(* Which data to send *)
				Server.UdpSend_0.datalen := SIZEOF(Server.data_buffer);	(* Lenght of data to send *)
				Server.UdpSend_0.flags := 0;
				Server.UdpSend_0;	(* Call the Function*)

				// Processing the received data
				packet.pStart				:= FIND(Server.data_buffer, 'pStart:');
				packet.pEnd					:= FIND(Server.data_buffer, 'pEnd');
				packet.length				:= UDINT_TO_INT(Server.UdpSend_0.datalen);
				packet.packet_pressure		:= MID(Server.data_buffer, packet.pEnd - packet.pStart-7, packet.pStart+7);

				FOR i:=0 TO 7 BY 1 DO
					packet.comma			:= FIND(packet.packet_pressure, ',');
					packet.pressureString[i]:= MID(packet.packet_pressure, packet.comma, 0);
					packet.packet_pressure	:= DELETE(packet.packet_pressure, packet.comma+1, 0);
					packet.pressureAO[i]	:= atof(ADR(packet.pressureString[i]));
				END_FOR

				IF Server.UdpSend_0.status = 0 THEN  (* Data sent *)
					Server.sStep := 1;
				ELSIF Server.UdpSend_0.status = ERR_FUB_BUSY THEN  (* UdpSend not finished -> redo *)
				  (* Busy *)
				ELSE  (* Goto Error Step *)
					Server.sStep := 10;
				END_IF

			10:  (* Here some error Handling has to be implemented *)

		END_CASE

	END_IF

END_PROGRAM
```

- Visualisation Logical/Visu (not shown)

### Program Logical/Riadenie/Program

#### Cyclic.st
```iecst
PROGRAM _CYCLIC

	IF zapni=TRUE THEN

	ELSE
		ventil_a1:=FALSE;
		ventil_b2:=FALSE;
		ventil_c3:=FALSE;
		ventil_d4:=FALSE;
	END_IF

END_PROGRAM
```

Listed in the project but not available here: Logical/Libraries/pomoc_lib/cyklovac_BB.c, Logical/Libraries/pomoc_lib/cyklovac_BB.h, Logical/Libraries/pomoc_lib/cyklovac_BB_data.c, Logical/Libraries/pomoc_lib/cyklovac_BB_types.h, Logical/Libraries/pomoc_lib/multiword_types.h, Logical/Libraries/pomoc_lib/pomoc_lib.fun, Logical/Libraries/pomoc_lib/pomoc_lib.var, Logical/Libraries/pomoc_lib/rtw_continuous.h, Logical/Libraries/pomoc_lib/rtw_solver.h, Logical/Libraries/pomoc_lib/tmwtypes.h, Logical/Libraries/regulatory/FF_PID_r_t.c, Logical/Libraries/regulatory/multiword_types.h, Logical/Libraries/regulatory/reg_FF_PI_pl_regr_stiff.c, Logical/Libraries/regulatory/regulatory.fun, Logical/Libraries/regulatory/regulatory.var, Logical/Libraries/regulatory/rtmodel.h, Logical/Libraries/regulatory/rtwtypes.h, Logical/Libraries/regulatory/PID_c.c, Logical/Libraries/regulatory/PID_co.c, Logical/Libraries/regulatory/PID_co.h, Logical/Libraries/regulatory/PID_co_private.h, Logical/Libraries/regulatory/PID_co_types.h, Logical/Libraries/regulatory/nonL_P.c, Logical/Libraries/regulatory/regulator_nelin_P.c, Logical/Libraries/regulatory/regulator_nelin_P.h, Logical/Libraries/regulatory/regulator_nelin_P_private.h, Logical/Libraries/regulatory/regulator_nelin_P_types.h, Logical/Libraries/regulatory/rt_defines.h, Logical/Libraries/regulatory/FF_PID_r.c, Logical/Libraries/regulatory/regulator_FF_PI_plane_regress.c, Logical/Libraries/regulatory/regulator_FF_PI_plane_regress.h, Logical/Libraries/regulatory/regulator_FF_PI_plane_regress_private.h, Logical/Libraries/regulatory/regulator_FF_PI_plane_regress_types.h, Logical/Libraries/regulatory/FF_PID.c, Logical/Libraries/regulatory/regulator_FF_PI.c, Logical/Libraries/regulatory/regulator_FF_PI.h, Logical/Libraries/regulatory/regulator_FF_PI_data.c, Logical/Libraries/regulatory/regulator_FF_PI_private.h, Logical/Libraries/regulatory/regulator_FF_PI_types.h, Logical/Libraries/regulatory/rtw_continuous.h, Logical/Libraries/regulatory/rtw_solver.h, Logical/Libraries/regulatory/tmwtypes.h
